// TIA Portal V17 export
// export: Created 2025-03-07T09:16:39.4097333Z, ExportSetting WithDefaults, DisplayName Totally Integrated Automation Portal, DisplayVersion V17 Update 8, DisplayName TIA Portal Openness, DisplayVersion V17 Update 8, DisplayName TIA Portal Version Control Interface, DisplayVersion V17, DisplayName SINAMICS Startdrive Advanced, DisplayVersion V17 SP2, DisplayName SINAMICS Startdrive G110M, G120, G120C, G120D, G120P, G115D, DisplayVersion V17 SP2, DisplayName SINAMICS Startdrive G130, G150, S120, S150, SINAMICS MV, S210, DisplayVersion V17 SP2, DisplayName STEP 7 Professional, DisplayVersion V17 Update 8, DisplayName SINUMERIK ONE STEP 7 Toolbox, DisplayVersion V17 Update 12, DisplayName SINUMERIK 840D sl STEP 7 Toolbox, DisplayVersion V17 Update 12, DisplayName STEP 7 Safety, DisplayVersion V17 Update 6, DisplayName WinCC Advanced, DisplayVersion V17 Update 8
FUNCTION "FC2420_CNC_PLC_SIGNALS" : Void   // FC2420, LAD
TITLE = NCK Inputs
{ S7_Optimized_Access := 'FALSE' }
AUTHOR : ETXETAR
VERSION : 1.0
// stored: AutoNumber false, IsIECCheckEnabled false, SetENOAutomatically false, UDAEnableTagReadback false
   VAR_TEMP
      ERROR : Bool;   // ERROR
      RESET_SIGNALS : Bool;   // RESET NC TO PLC SIGNALS
      ERROR_CODE : Int;   // ERROR CODE
      ZERO : Int;   // ZERO
   END_VAR
   VAR CONSTANT
      READ : Byte := 16#3;   // READ
      WRITE : Byte := 16#4;   // WRITE
   END_VAR
   VAR_TEMP   // added for the SCL form of the ladder/FBD networks
      _w1 : Bool;
   END_VAR
BEGIN

REGION Network 1: ZERO
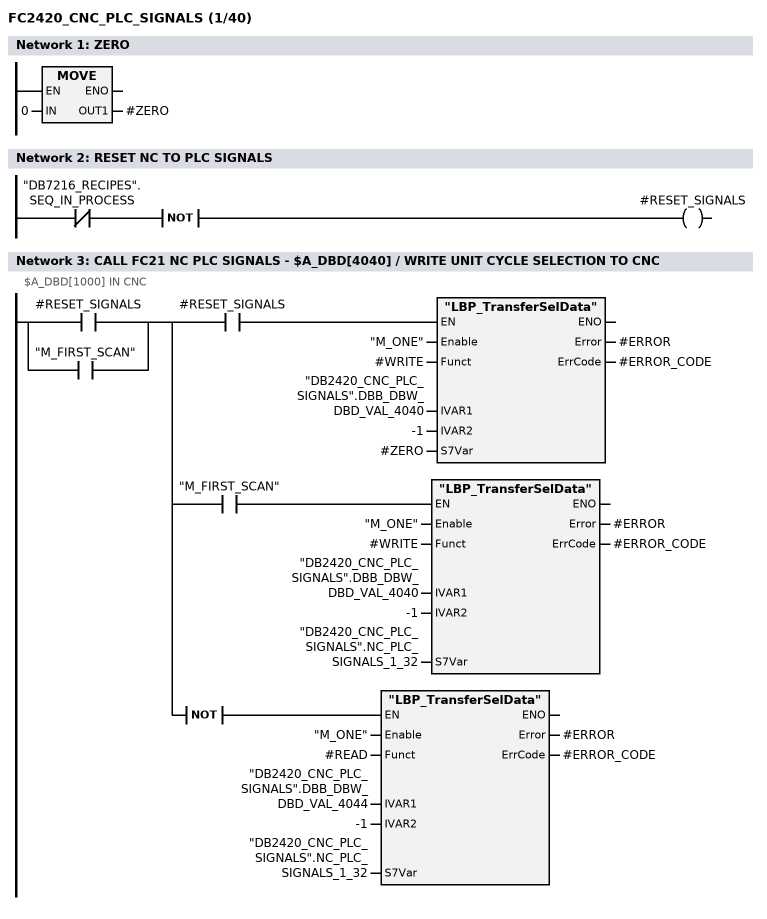
   RUNG wire#powerrail
      Move(in := 0, out1 => #ZERO)
   END_RUNG
   // the same network as SCL:
   #ZERO := 0;
END_REGION

REGION Network 2: RESET NC TO PLC SIGNALS
   RUNG wire#powerrail
      I_Contact( "DB7216_RECIPES".SEQ_IN_PROCESS )
      Not()
      Coil( #RESET_SIGNALS )
   END_RUNG
   // the same network as SCL:
   #RESET_SIGNALS := NOT (NOT "DB7216_RECIPES".SEQ_IN_PROCESS);
END_REGION

REGION Network 3: CALL FC21 NC PLC SIGNALS - $A_DBD[4040] / WRITE UNIT CYCLE SELECTION TO CNC
   // $A_DBD[1000] IN CNC
   RUNG wire#powerrail
      Contact( #RESET_SIGNALS )
      wire#w1
      Contact( #RESET_SIGNALS )
      "LBP_TransferSelData"(Enable := "M_ONE", Funct := #WRITE, IVAR1 := "DB2420_CNC_PLC_SIGNALS".DBB_DBW_DBD_VAL_4040, IVAR2 := -1, S7Var := #ZERO, Error => #ERROR, ErrCode => #ERROR_CODE)
   END_RUNG
   RUNG wire#powerrail
      Contact( "M_FIRST_SCAN" )
   END_RUNG wire#w1
   RUNG wire#w1
      Contact( "M_FIRST_SCAN" )
      "LBP_TransferSelData"(Enable := "M_ONE", Funct := #WRITE, IVAR1 := "DB2420_CNC_PLC_SIGNALS".DBB_DBW_DBD_VAL_4040, IVAR2 := -1, S7Var := "DB2420_CNC_PLC_SIGNALS".NC_PLC_SIGNALS_1_32, Error => #ERROR, ErrCode => #ERROR_CODE)
   END_RUNG
   RUNG wire#w1
      Not()
      "LBP_TransferSelData"(Enable := "M_ONE", Funct := #READ, IVAR1 := "DB2420_CNC_PLC_SIGNALS".DBB_DBW_DBD_VAL_4044, IVAR2 := -1, S7Var := "DB2420_CNC_PLC_SIGNALS".NC_PLC_SIGNALS_1_32, Error => #ERROR, ErrCode => #ERROR_CODE)
   END_RUNG
   // the same network as SCL:
   #_w1 := #RESET_SIGNALS OR "M_FIRST_SCAN";
   IF #_w1 AND #RESET_SIGNALS THEN
       "LBP_TransferSelData"(Enable := "M_ONE",
                             Funct := #WRITE,
                             IVAR1 := "DB2420_CNC_PLC_SIGNALS".DBB_DBW_DBD_VAL_4040,
                             IVAR2 := -1,
                             S7Var := #ZERO,
                             Error => #ERROR,
                             ErrCode => #ERROR_CODE);
   END_IF;
   IF #_w1 AND "M_FIRST_SCAN" THEN
       "LBP_TransferSelData"(Enable := "M_ONE",
                             Funct := #WRITE,
                             IVAR1 := "DB2420_CNC_PLC_SIGNALS".DBB_DBW_DBD_VAL_4040,
                             IVAR2 := -1,
                             S7Var := "DB2420_CNC_PLC_SIGNALS".NC_PLC_SIGNALS_1_32,
                             Error => #ERROR,
                             ErrCode => #ERROR_CODE);
   END_IF;
   IF NOT #_w1 THEN
       "LBP_TransferSelData"(Enable := "M_ONE",
                             Funct := #READ,
                             IVAR1 := "DB2420_CNC_PLC_SIGNALS".DBB_DBW_DBD_VAL_4044,
                             IVAR2 := -1,
                             S7Var := "DB2420_CNC_PLC_SIGNALS".NC_PLC_SIGNALS_1_32,
                             Error => #ERROR,
                             ErrCode => #ERROR_CODE);
   END_IF;
END_REGION

REGION Network 4: NC PLC SIGNALS 1-8
   // SIGNAL 1 -->  FIXTURE 1 CYLINDER 1 CLAMPED
   // SIGNAL 2 -->  FIXTURE 1 CYLINDER 2 CLAMPED
   // SIGNAL 3 -->  FIXTURE 1 CYLINDER 3 CLAMPED
   // SIGNAL 4 -->  FIXTURE 1 CYLINDER 4 CLAMPED
   // SIGNAL 5 -->  FIXTURE 1 CYLINDER 5 CLAMPED
   // SIGNAL 6 -->  FIXTURE 1 CYLINDER 6 CLAMPED
   // SIGNAL 7 -->  FIXTURE 1 CYLINDER 7 CLAMPED
   // SIGNAL 8 -->  FIXTURE 1 CYLINDER 8 CLAMPED
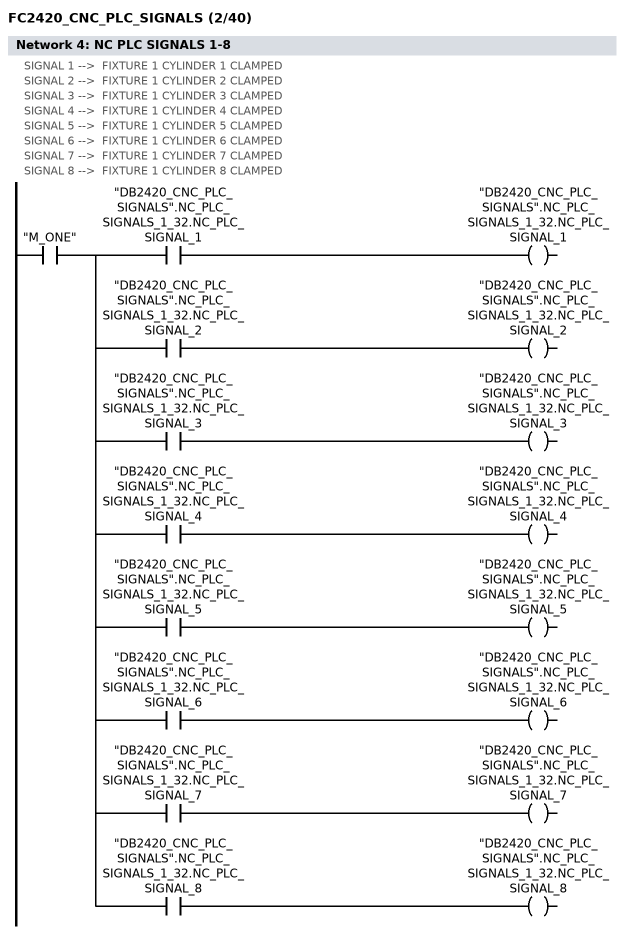
   RUNG wire#powerrail
      Contact( "M_ONE" )
      wire#w1
      Contact( "DB2420_CNC_PLC_SIGNALS".NC_PLC_SIGNALS_1_32.NC_PLC_SIGNAL_1 )
      Coil( "DB2420_CNC_PLC_SIGNALS".NC_PLC_SIGNALS_1_32.NC_PLC_SIGNAL_1 )
   END_RUNG
   RUNG wire#w1
      Contact( "DB2420_CNC_PLC_SIGNALS".NC_PLC_SIGNALS_1_32.NC_PLC_SIGNAL_2 )
      Coil( "DB2420_CNC_PLC_SIGNALS".NC_PLC_SIGNALS_1_32.NC_PLC_SIGNAL_2 )
   END_RUNG
   RUNG wire#w1
      Contact( "DB2420_CNC_PLC_SIGNALS".NC_PLC_SIGNALS_1_32.NC_PLC_SIGNAL_3 )
      Coil( "DB2420_CNC_PLC_SIGNALS".NC_PLC_SIGNALS_1_32.NC_PLC_SIGNAL_3 )
   END_RUNG
   RUNG wire#w1
      Contact( "DB2420_CNC_PLC_SIGNALS".NC_PLC_SIGNALS_1_32.NC_PLC_SIGNAL_4 )
      Coil( "DB2420_CNC_PLC_SIGNALS".NC_PLC_SIGNALS_1_32.NC_PLC_SIGNAL_4 )
   END_RUNG
   RUNG wire#w1
      Contact( "DB2420_CNC_PLC_SIGNALS".NC_PLC_SIGNALS_1_32.NC_PLC_SIGNAL_5 )
      Coil( "DB2420_CNC_PLC_SIGNALS".NC_PLC_SIGNALS_1_32.NC_PLC_SIGNAL_5 )
   END_RUNG
   RUNG wire#w1
      Contact( "DB2420_CNC_PLC_SIGNALS".NC_PLC_SIGNALS_1_32.NC_PLC_SIGNAL_6 )
      Coil( "DB2420_CNC_PLC_SIGNALS".NC_PLC_SIGNALS_1_32.NC_PLC_SIGNAL_6 )
   END_RUNG
   RUNG wire#w1
      Contact( "DB2420_CNC_PLC_SIGNALS".NC_PLC_SIGNALS_1_32.NC_PLC_SIGNAL_7 )
      Coil( "DB2420_CNC_PLC_SIGNALS".NC_PLC_SIGNALS_1_32.NC_PLC_SIGNAL_7 )
   END_RUNG
   RUNG wire#w1
      Contact( "DB2420_CNC_PLC_SIGNALS".NC_PLC_SIGNALS_1_32.NC_PLC_SIGNAL_8 )
      Coil( "DB2420_CNC_PLC_SIGNALS".NC_PLC_SIGNALS_1_32.NC_PLC_SIGNAL_8 )
   END_RUNG
   // the same network as SCL:
   "DB2420_CNC_PLC_SIGNALS".NC_PLC_SIGNALS_1_32.NC_PLC_SIGNAL_1 := "M_ONE" AND "DB2420_CNC_PLC_SIGNALS".NC_PLC_SIGNALS_1_32.NC_PLC_SIGNAL_1;
   "DB2420_CNC_PLC_SIGNALS".NC_PLC_SIGNALS_1_32.NC_PLC_SIGNAL_2 := "M_ONE" AND "DB2420_CNC_PLC_SIGNALS".NC_PLC_SIGNALS_1_32.NC_PLC_SIGNAL_2;
   "DB2420_CNC_PLC_SIGNALS".NC_PLC_SIGNALS_1_32.NC_PLC_SIGNAL_3 := "M_ONE" AND "DB2420_CNC_PLC_SIGNALS".NC_PLC_SIGNALS_1_32.NC_PLC_SIGNAL_3;
   "DB2420_CNC_PLC_SIGNALS".NC_PLC_SIGNALS_1_32.NC_PLC_SIGNAL_4 := "M_ONE" AND "DB2420_CNC_PLC_SIGNALS".NC_PLC_SIGNALS_1_32.NC_PLC_SIGNAL_4;
   "DB2420_CNC_PLC_SIGNALS".NC_PLC_SIGNALS_1_32.NC_PLC_SIGNAL_5 := "M_ONE" AND "DB2420_CNC_PLC_SIGNALS".NC_PLC_SIGNALS_1_32.NC_PLC_SIGNAL_5;
   "DB2420_CNC_PLC_SIGNALS".NC_PLC_SIGNALS_1_32.NC_PLC_SIGNAL_6 := "M_ONE" AND "DB2420_CNC_PLC_SIGNALS".NC_PLC_SIGNALS_1_32.NC_PLC_SIGNAL_6;
   "DB2420_CNC_PLC_SIGNALS".NC_PLC_SIGNALS_1_32.NC_PLC_SIGNAL_7 := "M_ONE" AND "DB2420_CNC_PLC_SIGNALS".NC_PLC_SIGNALS_1_32.NC_PLC_SIGNAL_7;
   "DB2420_CNC_PLC_SIGNALS".NC_PLC_SIGNALS_1_32.NC_PLC_SIGNAL_8 := "M_ONE" AND "DB2420_CNC_PLC_SIGNALS".NC_PLC_SIGNALS_1_32.NC_PLC_SIGNAL_8;
END_REGION

REGION Network 5: NC PLC SIGNALS 9-16
   // SIGNAL 9 -->  FIXTURE 1 CYLINDER 9 CLAMPED
   // SIGNAL 10 -->  FIXTURE 1 CYLINDER 10 CLAMPED
   // SIGNAL 11 -->  FIXTURE 1 CYLINDER 11 CLAMPED
   // SIGNAL 12 -->  FIXTURE 1 CYLINDER 12 CLAMPED
   // SIGNAL 13 -->  FIXTURE 1 CYLINDER 13 CLAMPED
   // SIGNAL 14 -->  FIXTURE 1 CYLINDER 14 CLAMPED
   // SIGNAL 15 -->  FIXTURE 1 CYLINDER 15 CLAMPED
   // SIGNAL 16 -->  FIXTURE 1 CYLINDER 16 CLAMPED
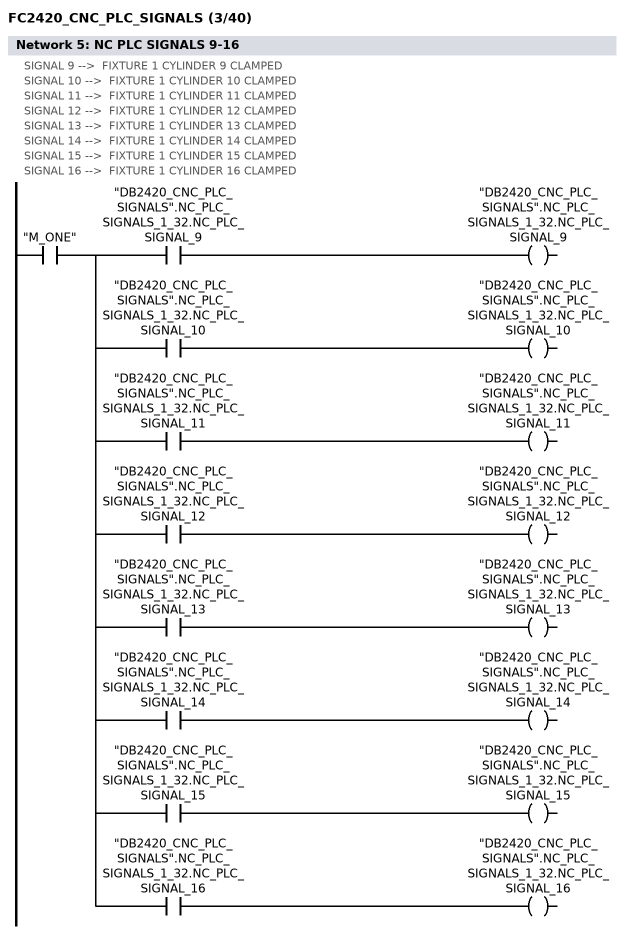
   RUNG wire#powerrail
      Contact( "M_ONE" )
      wire#w1
      Contact( "DB2420_CNC_PLC_SIGNALS".NC_PLC_SIGNALS_1_32.NC_PLC_SIGNAL_9 )
      Coil( "DB2420_CNC_PLC_SIGNALS".NC_PLC_SIGNALS_1_32.NC_PLC_SIGNAL_9 )
   END_RUNG
   RUNG wire#w1
      Contact( "DB2420_CNC_PLC_SIGNALS".NC_PLC_SIGNALS_1_32.NC_PLC_SIGNAL_10 )
      Coil( "DB2420_CNC_PLC_SIGNALS".NC_PLC_SIGNALS_1_32.NC_PLC_SIGNAL_10 )
   END_RUNG
   RUNG wire#w1
      Contact( "DB2420_CNC_PLC_SIGNALS".NC_PLC_SIGNALS_1_32.NC_PLC_SIGNAL_11 )
      Coil( "DB2420_CNC_PLC_SIGNALS".NC_PLC_SIGNALS_1_32.NC_PLC_SIGNAL_11 )
   END_RUNG
   RUNG wire#w1
      Contact( "DB2420_CNC_PLC_SIGNALS".NC_PLC_SIGNALS_1_32.NC_PLC_SIGNAL_12 )
      Coil( "DB2420_CNC_PLC_SIGNALS".NC_PLC_SIGNALS_1_32.NC_PLC_SIGNAL_12 )
   END_RUNG
   RUNG wire#w1
      Contact( "DB2420_CNC_PLC_SIGNALS".NC_PLC_SIGNALS_1_32.NC_PLC_SIGNAL_13 )
      Coil( "DB2420_CNC_PLC_SIGNALS".NC_PLC_SIGNALS_1_32.NC_PLC_SIGNAL_13 )
   END_RUNG
   RUNG wire#w1
      Contact( "DB2420_CNC_PLC_SIGNALS".NC_PLC_SIGNALS_1_32.NC_PLC_SIGNAL_14 )
      Coil( "DB2420_CNC_PLC_SIGNALS".NC_PLC_SIGNALS_1_32.NC_PLC_SIGNAL_14 )
   END_RUNG
   RUNG wire#w1
      Contact( "DB2420_CNC_PLC_SIGNALS".NC_PLC_SIGNALS_1_32.NC_PLC_SIGNAL_15 )
      Coil( "DB2420_CNC_PLC_SIGNALS".NC_PLC_SIGNALS_1_32.NC_PLC_SIGNAL_15 )
   END_RUNG
   RUNG wire#w1
      Contact( "DB2420_CNC_PLC_SIGNALS".NC_PLC_SIGNALS_1_32.NC_PLC_SIGNAL_16 )
      Coil( "DB2420_CNC_PLC_SIGNALS".NC_PLC_SIGNALS_1_32.NC_PLC_SIGNAL_16 )
   END_RUNG
   // the same network as SCL:
   "DB2420_CNC_PLC_SIGNALS".NC_PLC_SIGNALS_1_32.NC_PLC_SIGNAL_9 := "M_ONE" AND "DB2420_CNC_PLC_SIGNALS".NC_PLC_SIGNALS_1_32.NC_PLC_SIGNAL_9;
   "DB2420_CNC_PLC_SIGNALS".NC_PLC_SIGNALS_1_32.NC_PLC_SIGNAL_10 := "M_ONE" AND "DB2420_CNC_PLC_SIGNALS".NC_PLC_SIGNALS_1_32.NC_PLC_SIGNAL_10;
   "DB2420_CNC_PLC_SIGNALS".NC_PLC_SIGNALS_1_32.NC_PLC_SIGNAL_11 := "M_ONE" AND "DB2420_CNC_PLC_SIGNALS".NC_PLC_SIGNALS_1_32.NC_PLC_SIGNAL_11;
   "DB2420_CNC_PLC_SIGNALS".NC_PLC_SIGNALS_1_32.NC_PLC_SIGNAL_12 := "M_ONE" AND "DB2420_CNC_PLC_SIGNALS".NC_PLC_SIGNALS_1_32.NC_PLC_SIGNAL_12;
   "DB2420_CNC_PLC_SIGNALS".NC_PLC_SIGNALS_1_32.NC_PLC_SIGNAL_13 := "M_ONE" AND "DB2420_CNC_PLC_SIGNALS".NC_PLC_SIGNALS_1_32.NC_PLC_SIGNAL_13;
   "DB2420_CNC_PLC_SIGNALS".NC_PLC_SIGNALS_1_32.NC_PLC_SIGNAL_14 := "M_ONE" AND "DB2420_CNC_PLC_SIGNALS".NC_PLC_SIGNALS_1_32.NC_PLC_SIGNAL_14;
   "DB2420_CNC_PLC_SIGNALS".NC_PLC_SIGNALS_1_32.NC_PLC_SIGNAL_15 := "M_ONE" AND "DB2420_CNC_PLC_SIGNALS".NC_PLC_SIGNALS_1_32.NC_PLC_SIGNAL_15;
   "DB2420_CNC_PLC_SIGNALS".NC_PLC_SIGNALS_1_32.NC_PLC_SIGNAL_16 := "M_ONE" AND "DB2420_CNC_PLC_SIGNALS".NC_PLC_SIGNALS_1_32.NC_PLC_SIGNAL_16;
END_REGION

REGION Network 6: NC PLC SIGNALS 17-24
   // SIGNAL 17 -->  FIXTURE 1 CYLINDER 17 CLAMPED
   // SIGNAL 18 -->  FIXTURE 1 CYLINDER 18 CLAMPED
   // SIGNAL 19 -->  FIXTURE 1 CYLINDER 19 CLAMPED
   // SIGNAL 20 -->  FIXTURE 1 CYLINDER 20 CLAMPED
   // SIGNAL 21 -->  FIXTURE 1 CYLINDER 21 CLAMPED
   // SIGNAL 22 -->  FIXTURE 1 CYLINDER 22 CLAMPED
   // SIGNAL 23 -->  FIXTURE 1 CYLINDER 23 CLAMPED
   // SIGNAL 24 -->  FIXTURE 1 CYLINDER 24 CLAMPED
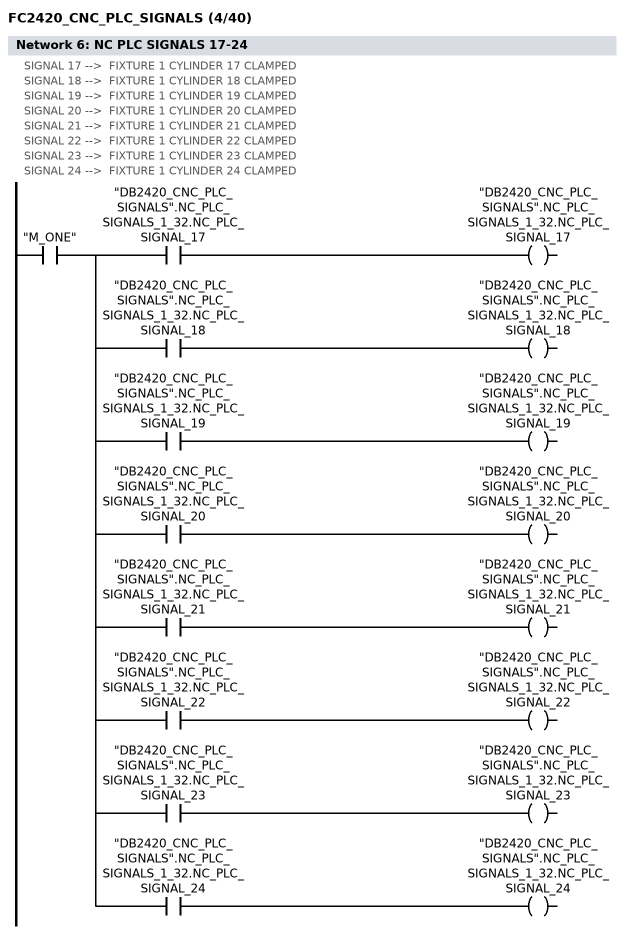
   RUNG wire#powerrail
      Contact( "M_ONE" )
      wire#w1
      Contact( "DB2420_CNC_PLC_SIGNALS".NC_PLC_SIGNALS_1_32.NC_PLC_SIGNAL_17 )
      Coil( "DB2420_CNC_PLC_SIGNALS".NC_PLC_SIGNALS_1_32.NC_PLC_SIGNAL_17 )
   END_RUNG
   RUNG wire#w1
      Contact( "DB2420_CNC_PLC_SIGNALS".NC_PLC_SIGNALS_1_32.NC_PLC_SIGNAL_18 )
      Coil( "DB2420_CNC_PLC_SIGNALS".NC_PLC_SIGNALS_1_32.NC_PLC_SIGNAL_18 )
   END_RUNG
   RUNG wire#w1
      Contact( "DB2420_CNC_PLC_SIGNALS".NC_PLC_SIGNALS_1_32.NC_PLC_SIGNAL_19 )
      Coil( "DB2420_CNC_PLC_SIGNALS".NC_PLC_SIGNALS_1_32.NC_PLC_SIGNAL_19 )
   END_RUNG
   RUNG wire#w1
      Contact( "DB2420_CNC_PLC_SIGNALS".NC_PLC_SIGNALS_1_32.NC_PLC_SIGNAL_20 )
      Coil( "DB2420_CNC_PLC_SIGNALS".NC_PLC_SIGNALS_1_32.NC_PLC_SIGNAL_20 )
   END_RUNG
   RUNG wire#w1
      Contact( "DB2420_CNC_PLC_SIGNALS".NC_PLC_SIGNALS_1_32.NC_PLC_SIGNAL_21 )
      Coil( "DB2420_CNC_PLC_SIGNALS".NC_PLC_SIGNALS_1_32.NC_PLC_SIGNAL_21 )
   END_RUNG
   RUNG wire#w1
      Contact( "DB2420_CNC_PLC_SIGNALS".NC_PLC_SIGNALS_1_32.NC_PLC_SIGNAL_22 )
      Coil( "DB2420_CNC_PLC_SIGNALS".NC_PLC_SIGNALS_1_32.NC_PLC_SIGNAL_22 )
   END_RUNG
   RUNG wire#w1
      Contact( "DB2420_CNC_PLC_SIGNALS".NC_PLC_SIGNALS_1_32.NC_PLC_SIGNAL_23 )
      Coil( "DB2420_CNC_PLC_SIGNALS".NC_PLC_SIGNALS_1_32.NC_PLC_SIGNAL_23 )
   END_RUNG
   RUNG wire#w1
      Contact( "DB2420_CNC_PLC_SIGNALS".NC_PLC_SIGNALS_1_32.NC_PLC_SIGNAL_24 )
      Coil( "DB2420_CNC_PLC_SIGNALS".NC_PLC_SIGNALS_1_32.NC_PLC_SIGNAL_24 )
   END_RUNG
   // the same network as SCL:
   "DB2420_CNC_PLC_SIGNALS".NC_PLC_SIGNALS_1_32.NC_PLC_SIGNAL_17 := "M_ONE" AND "DB2420_CNC_PLC_SIGNALS".NC_PLC_SIGNALS_1_32.NC_PLC_SIGNAL_17;
   "DB2420_CNC_PLC_SIGNALS".NC_PLC_SIGNALS_1_32.NC_PLC_SIGNAL_18 := "M_ONE" AND "DB2420_CNC_PLC_SIGNALS".NC_PLC_SIGNALS_1_32.NC_PLC_SIGNAL_18;
   "DB2420_CNC_PLC_SIGNALS".NC_PLC_SIGNALS_1_32.NC_PLC_SIGNAL_19 := "M_ONE" AND "DB2420_CNC_PLC_SIGNALS".NC_PLC_SIGNALS_1_32.NC_PLC_SIGNAL_19;
   "DB2420_CNC_PLC_SIGNALS".NC_PLC_SIGNALS_1_32.NC_PLC_SIGNAL_20 := "M_ONE" AND "DB2420_CNC_PLC_SIGNALS".NC_PLC_SIGNALS_1_32.NC_PLC_SIGNAL_20;
   "DB2420_CNC_PLC_SIGNALS".NC_PLC_SIGNALS_1_32.NC_PLC_SIGNAL_21 := "M_ONE" AND "DB2420_CNC_PLC_SIGNALS".NC_PLC_SIGNALS_1_32.NC_PLC_SIGNAL_21;
   "DB2420_CNC_PLC_SIGNALS".NC_PLC_SIGNALS_1_32.NC_PLC_SIGNAL_22 := "M_ONE" AND "DB2420_CNC_PLC_SIGNALS".NC_PLC_SIGNALS_1_32.NC_PLC_SIGNAL_22;
   "DB2420_CNC_PLC_SIGNALS".NC_PLC_SIGNALS_1_32.NC_PLC_SIGNAL_23 := "M_ONE" AND "DB2420_CNC_PLC_SIGNALS".NC_PLC_SIGNALS_1_32.NC_PLC_SIGNAL_23;
   "DB2420_CNC_PLC_SIGNALS".NC_PLC_SIGNALS_1_32.NC_PLC_SIGNAL_24 := "M_ONE" AND "DB2420_CNC_PLC_SIGNALS".NC_PLC_SIGNALS_1_32.NC_PLC_SIGNAL_24;
END_REGION

REGION Network 7: NC PLC SIGNALS 25-32
   // SIGNAL 25 -->  FIXTURE 1 CYLINDER 1 UNCLAMPED
   // SIGNAL 26 -->  FIXTURE 1 CYLINDER 2 UNCLAMPED
   // SIGNAL 27 -->  FIXTURE 1 CYLINDER 3 UNCLAMPED
   // SIGNAL 28 -->  FIXTURE 1 CYLINDER 4 UNCLAMPED
   // SIGNAL 29 -->  FIXTURE 1 CYLINDER 5 UNCLAMPED
   // SIGNAL 30 -->  FIXTURE 1 CYLINDER 6 UNCLAMPED
   // SIGNAL 31 -->  FIXTURE 1 CYLINDER 7 UNCLAMPED
   // SIGNAL 32 -->  FIXTURE 1 CYLINDER 8 UNCLAMPED
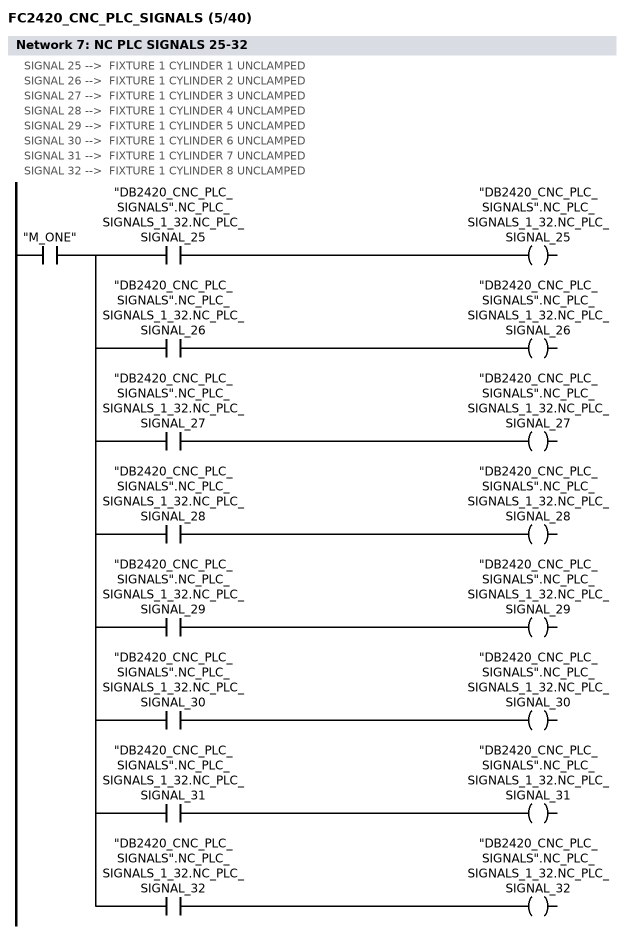
   RUNG wire#powerrail
      Contact( "M_ONE" )
      wire#w1
      Contact( "DB2420_CNC_PLC_SIGNALS".NC_PLC_SIGNALS_1_32.NC_PLC_SIGNAL_25 )
      Coil( "DB2420_CNC_PLC_SIGNALS".NC_PLC_SIGNALS_1_32.NC_PLC_SIGNAL_25 )
   END_RUNG
   RUNG wire#w1
      Contact( "DB2420_CNC_PLC_SIGNALS".NC_PLC_SIGNALS_1_32.NC_PLC_SIGNAL_26 )
      Coil( "DB2420_CNC_PLC_SIGNALS".NC_PLC_SIGNALS_1_32.NC_PLC_SIGNAL_26 )
   END_RUNG
   RUNG wire#w1
      Contact( "DB2420_CNC_PLC_SIGNALS".NC_PLC_SIGNALS_1_32.NC_PLC_SIGNAL_27 )
      Coil( "DB2420_CNC_PLC_SIGNALS".NC_PLC_SIGNALS_1_32.NC_PLC_SIGNAL_27 )
   END_RUNG
   RUNG wire#w1
      Contact( "DB2420_CNC_PLC_SIGNALS".NC_PLC_SIGNALS_1_32.NC_PLC_SIGNAL_28 )
      Coil( "DB2420_CNC_PLC_SIGNALS".NC_PLC_SIGNALS_1_32.NC_PLC_SIGNAL_28 )
   END_RUNG
   RUNG wire#w1
      Contact( "DB2420_CNC_PLC_SIGNALS".NC_PLC_SIGNALS_1_32.NC_PLC_SIGNAL_29 )
      Coil( "DB2420_CNC_PLC_SIGNALS".NC_PLC_SIGNALS_1_32.NC_PLC_SIGNAL_29 )
   END_RUNG
   RUNG wire#w1
      Contact( "DB2420_CNC_PLC_SIGNALS".NC_PLC_SIGNALS_1_32.NC_PLC_SIGNAL_30 )
      Coil( "DB2420_CNC_PLC_SIGNALS".NC_PLC_SIGNALS_1_32.NC_PLC_SIGNAL_30 )
   END_RUNG
   RUNG wire#w1
      Contact( "DB2420_CNC_PLC_SIGNALS".NC_PLC_SIGNALS_1_32.NC_PLC_SIGNAL_31 )
      Coil( "DB2420_CNC_PLC_SIGNALS".NC_PLC_SIGNALS_1_32.NC_PLC_SIGNAL_31 )
   END_RUNG
   RUNG wire#w1
      Contact( "DB2420_CNC_PLC_SIGNALS".NC_PLC_SIGNALS_1_32.NC_PLC_SIGNAL_32 )
      Coil( "DB2420_CNC_PLC_SIGNALS".NC_PLC_SIGNALS_1_32.NC_PLC_SIGNAL_32 )
   END_RUNG
   // the same network as SCL:
   "DB2420_CNC_PLC_SIGNALS".NC_PLC_SIGNALS_1_32.NC_PLC_SIGNAL_25 := "M_ONE" AND "DB2420_CNC_PLC_SIGNALS".NC_PLC_SIGNALS_1_32.NC_PLC_SIGNAL_25;
   "DB2420_CNC_PLC_SIGNALS".NC_PLC_SIGNALS_1_32.NC_PLC_SIGNAL_26 := "M_ONE" AND "DB2420_CNC_PLC_SIGNALS".NC_PLC_SIGNALS_1_32.NC_PLC_SIGNAL_26;
   "DB2420_CNC_PLC_SIGNALS".NC_PLC_SIGNALS_1_32.NC_PLC_SIGNAL_27 := "M_ONE" AND "DB2420_CNC_PLC_SIGNALS".NC_PLC_SIGNALS_1_32.NC_PLC_SIGNAL_27;
   "DB2420_CNC_PLC_SIGNALS".NC_PLC_SIGNALS_1_32.NC_PLC_SIGNAL_28 := "M_ONE" AND "DB2420_CNC_PLC_SIGNALS".NC_PLC_SIGNALS_1_32.NC_PLC_SIGNAL_28;
   "DB2420_CNC_PLC_SIGNALS".NC_PLC_SIGNALS_1_32.NC_PLC_SIGNAL_29 := "M_ONE" AND "DB2420_CNC_PLC_SIGNALS".NC_PLC_SIGNALS_1_32.NC_PLC_SIGNAL_29;
   "DB2420_CNC_PLC_SIGNALS".NC_PLC_SIGNALS_1_32.NC_PLC_SIGNAL_30 := "M_ONE" AND "DB2420_CNC_PLC_SIGNALS".NC_PLC_SIGNALS_1_32.NC_PLC_SIGNAL_30;
   "DB2420_CNC_PLC_SIGNALS".NC_PLC_SIGNALS_1_32.NC_PLC_SIGNAL_31 := "M_ONE" AND "DB2420_CNC_PLC_SIGNALS".NC_PLC_SIGNALS_1_32.NC_PLC_SIGNAL_31;
   "DB2420_CNC_PLC_SIGNALS".NC_PLC_SIGNALS_1_32.NC_PLC_SIGNAL_32 := "M_ONE" AND "DB2420_CNC_PLC_SIGNALS".NC_PLC_SIGNALS_1_32.NC_PLC_SIGNAL_32;
END_REGION

REGION Network 8: CALL FC21 NC PLC SIGNALS- $A_DBD[4044] / WRITE UNIT CYCLE SELECTION TO CNC
   // $A_DBD[1000] IN CNC
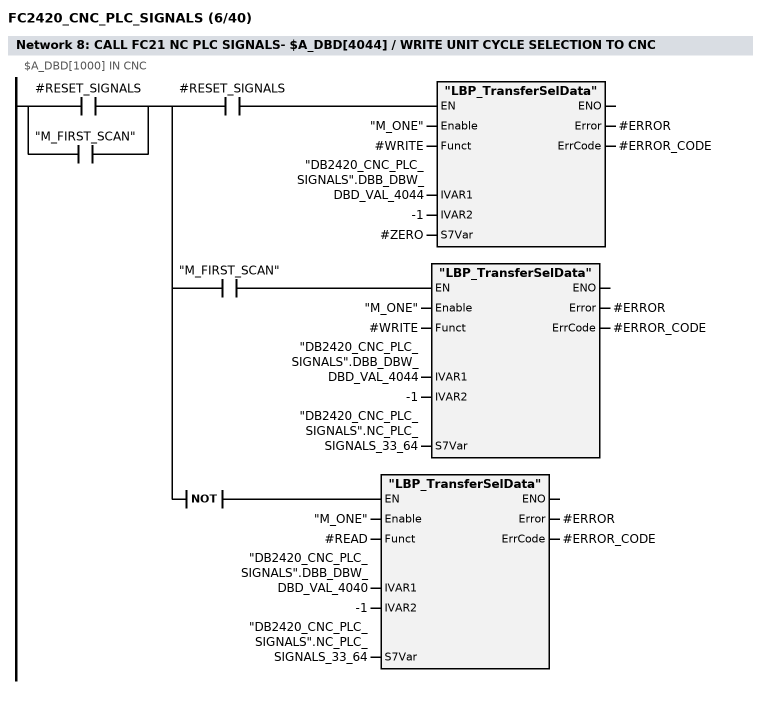
   RUNG wire#powerrail
      Contact( #RESET_SIGNALS )
      wire#w1
      Contact( #RESET_SIGNALS )
      "LBP_TransferSelData"(Enable := "M_ONE", Funct := #WRITE, IVAR1 := "DB2420_CNC_PLC_SIGNALS".DBB_DBW_DBD_VAL_4044, IVAR2 := -1, S7Var := #ZERO, Error => #ERROR, ErrCode => #ERROR_CODE)
   END_RUNG
   RUNG wire#powerrail
      Contact( "M_FIRST_SCAN" )
   END_RUNG wire#w1
   RUNG wire#w1
      Contact( "M_FIRST_SCAN" )
      "LBP_TransferSelData"(Enable := "M_ONE", Funct := #WRITE, IVAR1 := "DB2420_CNC_PLC_SIGNALS".DBB_DBW_DBD_VAL_4044, IVAR2 := -1, S7Var := "DB2420_CNC_PLC_SIGNALS".NC_PLC_SIGNALS_33_64, Error => #ERROR, ErrCode => #ERROR_CODE)
   END_RUNG
   RUNG wire#w1
      Not()
      "LBP_TransferSelData"(Enable := "M_ONE", Funct := #READ, IVAR1 := "DB2420_CNC_PLC_SIGNALS".DBB_DBW_DBD_VAL_4040, IVAR2 := -1, S7Var := "DB2420_CNC_PLC_SIGNALS".NC_PLC_SIGNALS_33_64, Error => #ERROR, ErrCode => #ERROR_CODE)
   END_RUNG
   // the same network as SCL:
   #_w1 := #RESET_SIGNALS OR "M_FIRST_SCAN";
   IF #_w1 AND #RESET_SIGNALS THEN
       "LBP_TransferSelData"(Enable := "M_ONE",
                             Funct := #WRITE,
                             IVAR1 := "DB2420_CNC_PLC_SIGNALS".DBB_DBW_DBD_VAL_4044,
                             IVAR2 := -1,
                             S7Var := #ZERO,
                             Error => #ERROR,
                             ErrCode => #ERROR_CODE);
   END_IF;
   IF #_w1 AND "M_FIRST_SCAN" THEN
       "LBP_TransferSelData"(Enable := "M_ONE",
                             Funct := #WRITE,
                             IVAR1 := "DB2420_CNC_PLC_SIGNALS".DBB_DBW_DBD_VAL_4044,
                             IVAR2 := -1,
                             S7Var := "DB2420_CNC_PLC_SIGNALS".NC_PLC_SIGNALS_33_64,
                             Error => #ERROR,
                             ErrCode => #ERROR_CODE);
   END_IF;
   IF NOT #_w1 THEN
       "LBP_TransferSelData"(Enable := "M_ONE",
                             Funct := #READ,
                             IVAR1 := "DB2420_CNC_PLC_SIGNALS".DBB_DBW_DBD_VAL_4040,
                             IVAR2 := -1,
                             S7Var := "DB2420_CNC_PLC_SIGNALS".NC_PLC_SIGNALS_33_64,
                             Error => #ERROR,
                             ErrCode => #ERROR_CODE);
   END_IF;
END_REGION

REGION Network 9: NC PLC SIGNALS 33-40
   // SIGNAL 33 -->  FIXTURE 1 CYLINDER 9 UNCLAMPED
   // SIGNAL 34 -->  FIXTURE 1 CYLINDER 10 UNCLAMPED
   // SIGNAL 35 -->  FIXTURE 1 CYLINDER 11 UNCLAMPED
   // SIGNAL 36 -->  FIXTURE 1 CYLINDER 12 UNCLAMPED
   // SIGNAL 37 -->  FIXTURE 1 CYLINDER 13 UNCLAMPED
   // SIGNAL 38 -->  FIXTURE 1 CYLINDER 14 UNCLAMPED
   // SIGNAL 39 -->  FIXTURE 1 CYLINDER 15 UNCLAMPED
   // SIGNAL 40 -->  FIXTURE 1 CYLINDER 16 UNCLAMPED
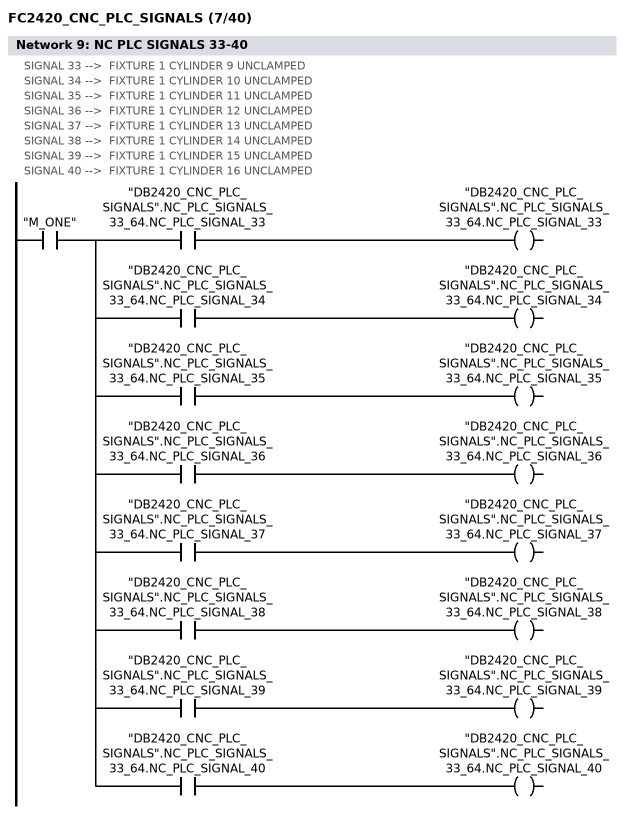
   RUNG wire#powerrail
      Contact( "M_ONE" )
      wire#w1
      Contact( "DB2420_CNC_PLC_SIGNALS".NC_PLC_SIGNALS_33_64.NC_PLC_SIGNAL_33 )
      Coil( "DB2420_CNC_PLC_SIGNALS".NC_PLC_SIGNALS_33_64.NC_PLC_SIGNAL_33 )
   END_RUNG
   RUNG wire#w1
      Contact( "DB2420_CNC_PLC_SIGNALS".NC_PLC_SIGNALS_33_64.NC_PLC_SIGNAL_34 )
      Coil( "DB2420_CNC_PLC_SIGNALS".NC_PLC_SIGNALS_33_64.NC_PLC_SIGNAL_34 )
   END_RUNG
   RUNG wire#w1
      Contact( "DB2420_CNC_PLC_SIGNALS".NC_PLC_SIGNALS_33_64.NC_PLC_SIGNAL_35 )
      Coil( "DB2420_CNC_PLC_SIGNALS".NC_PLC_SIGNALS_33_64.NC_PLC_SIGNAL_35 )
   END_RUNG
   RUNG wire#w1
      Contact( "DB2420_CNC_PLC_SIGNALS".NC_PLC_SIGNALS_33_64.NC_PLC_SIGNAL_36 )
      Coil( "DB2420_CNC_PLC_SIGNALS".NC_PLC_SIGNALS_33_64.NC_PLC_SIGNAL_36 )
   END_RUNG
   RUNG wire#w1
      Contact( "DB2420_CNC_PLC_SIGNALS".NC_PLC_SIGNALS_33_64.NC_PLC_SIGNAL_37 )
      Coil( "DB2420_CNC_PLC_SIGNALS".NC_PLC_SIGNALS_33_64.NC_PLC_SIGNAL_37 )
   END_RUNG
   RUNG wire#w1
      Contact( "DB2420_CNC_PLC_SIGNALS".NC_PLC_SIGNALS_33_64.NC_PLC_SIGNAL_38 )
      Coil( "DB2420_CNC_PLC_SIGNALS".NC_PLC_SIGNALS_33_64.NC_PLC_SIGNAL_38 )
   END_RUNG
   RUNG wire#w1
      Contact( "DB2420_CNC_PLC_SIGNALS".NC_PLC_SIGNALS_33_64.NC_PLC_SIGNAL_39 )
      Coil( "DB2420_CNC_PLC_SIGNALS".NC_PLC_SIGNALS_33_64.NC_PLC_SIGNAL_39 )
   END_RUNG
   RUNG wire#w1
      Contact( "DB2420_CNC_PLC_SIGNALS".NC_PLC_SIGNALS_33_64.NC_PLC_SIGNAL_40 )
      Coil( "DB2420_CNC_PLC_SIGNALS".NC_PLC_SIGNALS_33_64.NC_PLC_SIGNAL_40 )
   END_RUNG
   // the same network as SCL:
   "DB2420_CNC_PLC_SIGNALS".NC_PLC_SIGNALS_33_64.NC_PLC_SIGNAL_33 := "M_ONE" AND "DB2420_CNC_PLC_SIGNALS".NC_PLC_SIGNALS_33_64.NC_PLC_SIGNAL_33;
   "DB2420_CNC_PLC_SIGNALS".NC_PLC_SIGNALS_33_64.NC_PLC_SIGNAL_34 := "M_ONE" AND "DB2420_CNC_PLC_SIGNALS".NC_PLC_SIGNALS_33_64.NC_PLC_SIGNAL_34;
   "DB2420_CNC_PLC_SIGNALS".NC_PLC_SIGNALS_33_64.NC_PLC_SIGNAL_35 := "M_ONE" AND "DB2420_CNC_PLC_SIGNALS".NC_PLC_SIGNALS_33_64.NC_PLC_SIGNAL_35;
   "DB2420_CNC_PLC_SIGNALS".NC_PLC_SIGNALS_33_64.NC_PLC_SIGNAL_36 := "M_ONE" AND "DB2420_CNC_PLC_SIGNALS".NC_PLC_SIGNALS_33_64.NC_PLC_SIGNAL_36;
   "DB2420_CNC_PLC_SIGNALS".NC_PLC_SIGNALS_33_64.NC_PLC_SIGNAL_37 := "M_ONE" AND "DB2420_CNC_PLC_SIGNALS".NC_PLC_SIGNALS_33_64.NC_PLC_SIGNAL_37;
   "DB2420_CNC_PLC_SIGNALS".NC_PLC_SIGNALS_33_64.NC_PLC_SIGNAL_38 := "M_ONE" AND "DB2420_CNC_PLC_SIGNALS".NC_PLC_SIGNALS_33_64.NC_PLC_SIGNAL_38;
   "DB2420_CNC_PLC_SIGNALS".NC_PLC_SIGNALS_33_64.NC_PLC_SIGNAL_39 := "M_ONE" AND "DB2420_CNC_PLC_SIGNALS".NC_PLC_SIGNALS_33_64.NC_PLC_SIGNAL_39;
   "DB2420_CNC_PLC_SIGNALS".NC_PLC_SIGNALS_33_64.NC_PLC_SIGNAL_40 := "M_ONE" AND "DB2420_CNC_PLC_SIGNALS".NC_PLC_SIGNALS_33_64.NC_PLC_SIGNAL_40;
END_REGION

REGION Network 10: NC PLC SIGNALS 41-48
   // SIGNAL 41 -->  FIXTURE 1 CYLINDER 17 UNCLAMPED
   // SIGNAL 42 -->  FIXTURE 1 CYLINDER 18 UNCLAMPED
   // SIGNAL 43 -->  FIXTURE 1 CYLINDER 19 UNCLAMPED
   // SIGNAL 44 -->  FIXTURE 1 CYLINDER 20 UNCLAMPED
   // SIGNAL 45 -->  FIXTURE 1 CYLINDER 21 UNCLAMPED
   // SIGNAL 46 -->  FIXTURE 1 CYLINDER 22 UNCLAMPED
   // SIGNAL 47 -->  FIXTURE 1 CYLINDER 23 UNCLAMPED
   // SIGNAL 48 -->  FIXTURE 1 CYLINDER 24 UNCLAMPED
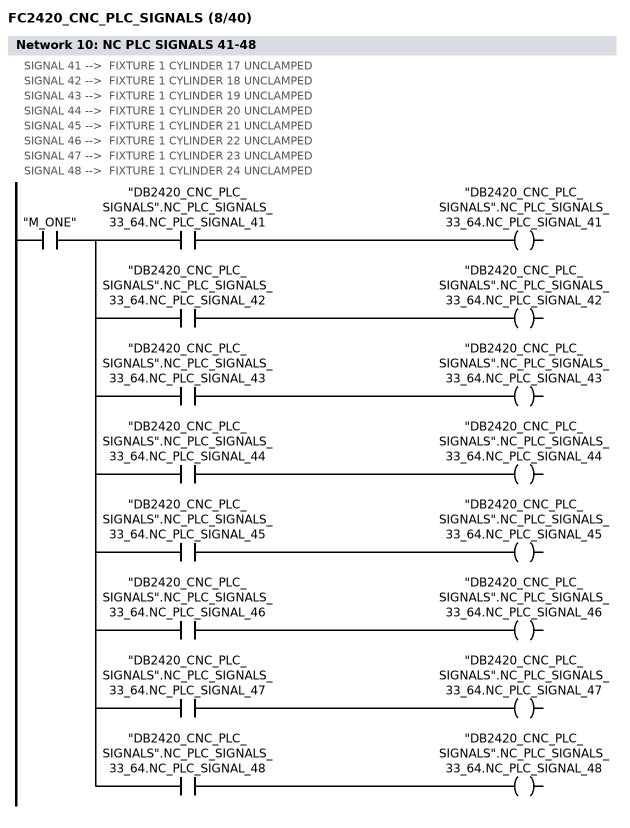
   RUNG wire#powerrail
      Contact( "M_ONE" )
      wire#w1
      Contact( "DB2420_CNC_PLC_SIGNALS".NC_PLC_SIGNALS_33_64.NC_PLC_SIGNAL_41 )
      Coil( "DB2420_CNC_PLC_SIGNALS".NC_PLC_SIGNALS_33_64.NC_PLC_SIGNAL_41 )
   END_RUNG
   RUNG wire#w1
      Contact( "DB2420_CNC_PLC_SIGNALS".NC_PLC_SIGNALS_33_64.NC_PLC_SIGNAL_42 )
      Coil( "DB2420_CNC_PLC_SIGNALS".NC_PLC_SIGNALS_33_64.NC_PLC_SIGNAL_42 )
   END_RUNG
   RUNG wire#w1
      Contact( "DB2420_CNC_PLC_SIGNALS".NC_PLC_SIGNALS_33_64.NC_PLC_SIGNAL_43 )
      Coil( "DB2420_CNC_PLC_SIGNALS".NC_PLC_SIGNALS_33_64.NC_PLC_SIGNAL_43 )
   END_RUNG
   RUNG wire#w1
      Contact( "DB2420_CNC_PLC_SIGNALS".NC_PLC_SIGNALS_33_64.NC_PLC_SIGNAL_44 )
      Coil( "DB2420_CNC_PLC_SIGNALS".NC_PLC_SIGNALS_33_64.NC_PLC_SIGNAL_44 )
   END_RUNG
   RUNG wire#w1
      Contact( "DB2420_CNC_PLC_SIGNALS".NC_PLC_SIGNALS_33_64.NC_PLC_SIGNAL_45 )
      Coil( "DB2420_CNC_PLC_SIGNALS".NC_PLC_SIGNALS_33_64.NC_PLC_SIGNAL_45 )
   END_RUNG
   RUNG wire#w1
      Contact( "DB2420_CNC_PLC_SIGNALS".NC_PLC_SIGNALS_33_64.NC_PLC_SIGNAL_46 )
      Coil( "DB2420_CNC_PLC_SIGNALS".NC_PLC_SIGNALS_33_64.NC_PLC_SIGNAL_46 )
   END_RUNG
   RUNG wire#w1
      Contact( "DB2420_CNC_PLC_SIGNALS".NC_PLC_SIGNALS_33_64.NC_PLC_SIGNAL_47 )
      Coil( "DB2420_CNC_PLC_SIGNALS".NC_PLC_SIGNALS_33_64.NC_PLC_SIGNAL_47 )
   END_RUNG
   RUNG wire#w1
      Contact( "DB2420_CNC_PLC_SIGNALS".NC_PLC_SIGNALS_33_64.NC_PLC_SIGNAL_48 )
      Coil( "DB2420_CNC_PLC_SIGNALS".NC_PLC_SIGNALS_33_64.NC_PLC_SIGNAL_48 )
   END_RUNG
   // the same network as SCL:
   "DB2420_CNC_PLC_SIGNALS".NC_PLC_SIGNALS_33_64.NC_PLC_SIGNAL_41 := "M_ONE" AND "DB2420_CNC_PLC_SIGNALS".NC_PLC_SIGNALS_33_64.NC_PLC_SIGNAL_41;
   "DB2420_CNC_PLC_SIGNALS".NC_PLC_SIGNALS_33_64.NC_PLC_SIGNAL_42 := "M_ONE" AND "DB2420_CNC_PLC_SIGNALS".NC_PLC_SIGNALS_33_64.NC_PLC_SIGNAL_42;
   "DB2420_CNC_PLC_SIGNALS".NC_PLC_SIGNALS_33_64.NC_PLC_SIGNAL_43 := "M_ONE" AND "DB2420_CNC_PLC_SIGNALS".NC_PLC_SIGNALS_33_64.NC_PLC_SIGNAL_43;
   "DB2420_CNC_PLC_SIGNALS".NC_PLC_SIGNALS_33_64.NC_PLC_SIGNAL_44 := "M_ONE" AND "DB2420_CNC_PLC_SIGNALS".NC_PLC_SIGNALS_33_64.NC_PLC_SIGNAL_44;
   "DB2420_CNC_PLC_SIGNALS".NC_PLC_SIGNALS_33_64.NC_PLC_SIGNAL_45 := "M_ONE" AND "DB2420_CNC_PLC_SIGNALS".NC_PLC_SIGNALS_33_64.NC_PLC_SIGNAL_45;
   "DB2420_CNC_PLC_SIGNALS".NC_PLC_SIGNALS_33_64.NC_PLC_SIGNAL_46 := "M_ONE" AND "DB2420_CNC_PLC_SIGNALS".NC_PLC_SIGNALS_33_64.NC_PLC_SIGNAL_46;
   "DB2420_CNC_PLC_SIGNALS".NC_PLC_SIGNALS_33_64.NC_PLC_SIGNAL_47 := "M_ONE" AND "DB2420_CNC_PLC_SIGNALS".NC_PLC_SIGNALS_33_64.NC_PLC_SIGNAL_47;
   "DB2420_CNC_PLC_SIGNALS".NC_PLC_SIGNALS_33_64.NC_PLC_SIGNAL_48 := "M_ONE" AND "DB2420_CNC_PLC_SIGNALS".NC_PLC_SIGNALS_33_64.NC_PLC_SIGNAL_48;
END_REGION

REGION Network 11: NC PLC SIGNALS 49-56
   // SIGNAL 49 -->  FIXTURE 2 CYLINDER 1 CLAMPED
   // SIGNAL 50 -->  FIXTURE 2 CYLINDER 2 CLAMPED
   // SIGNAL 51 -->   FIXTURE 2 CYLINDER 3 CLAMPED
   // SIGNAL 52 -->   FIXTURE 2 CYLINDER 4 CLAMPED
   // SIGNAL 53 -->   FIXTURE 2 CYLINDER 5 CLAMPED
   // SIGNAL 54 -->   FIXTURE 2 CYLINDER 6 CLAMPED
   // SIGNAL 55 -->   FIXTURE 2 CYLINDER 7 CLAMPED
   // SIGNAL 56 -->   FIXTURE 2 CYLINDER 8 CLAMPED
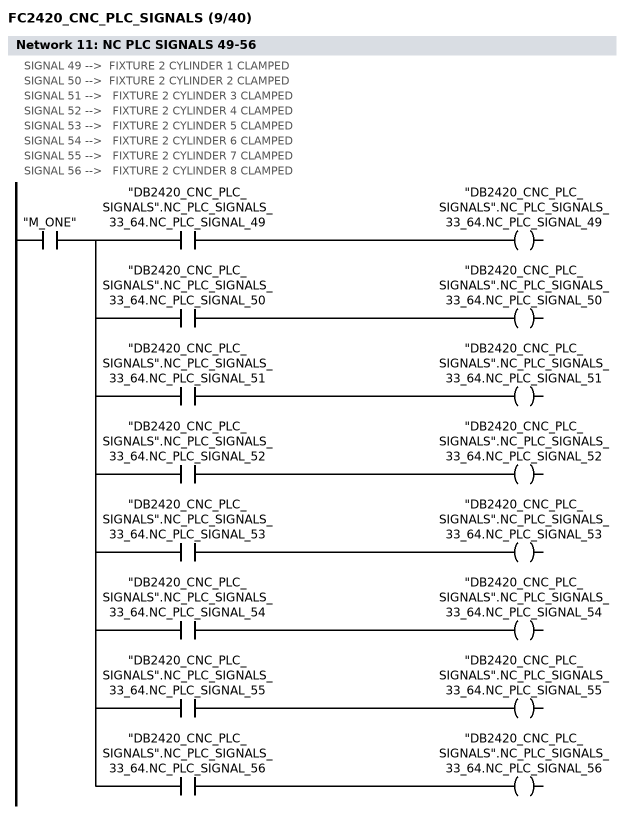
   RUNG wire#powerrail
      Contact( "M_ONE" )
      wire#w1
      Contact( "DB2420_CNC_PLC_SIGNALS".NC_PLC_SIGNALS_33_64.NC_PLC_SIGNAL_49 )
      Coil( "DB2420_CNC_PLC_SIGNALS".NC_PLC_SIGNALS_33_64.NC_PLC_SIGNAL_49 )
   END_RUNG
   RUNG wire#w1
      Contact( "DB2420_CNC_PLC_SIGNALS".NC_PLC_SIGNALS_33_64.NC_PLC_SIGNAL_50 )
      Coil( "DB2420_CNC_PLC_SIGNALS".NC_PLC_SIGNALS_33_64.NC_PLC_SIGNAL_50 )
   END_RUNG
   RUNG wire#w1
      Contact( "DB2420_CNC_PLC_SIGNALS".NC_PLC_SIGNALS_33_64.NC_PLC_SIGNAL_51 )
      Coil( "DB2420_CNC_PLC_SIGNALS".NC_PLC_SIGNALS_33_64.NC_PLC_SIGNAL_51 )
   END_RUNG
   RUNG wire#w1
      Contact( "DB2420_CNC_PLC_SIGNALS".NC_PLC_SIGNALS_33_64.NC_PLC_SIGNAL_52 )
      Coil( "DB2420_CNC_PLC_SIGNALS".NC_PLC_SIGNALS_33_64.NC_PLC_SIGNAL_52 )
   END_RUNG
   RUNG wire#w1
      Contact( "DB2420_CNC_PLC_SIGNALS".NC_PLC_SIGNALS_33_64.NC_PLC_SIGNAL_53 )
      Coil( "DB2420_CNC_PLC_SIGNALS".NC_PLC_SIGNALS_33_64.NC_PLC_SIGNAL_53 )
   END_RUNG
   RUNG wire#w1
      Contact( "DB2420_CNC_PLC_SIGNALS".NC_PLC_SIGNALS_33_64.NC_PLC_SIGNAL_54 )
      Coil( "DB2420_CNC_PLC_SIGNALS".NC_PLC_SIGNALS_33_64.NC_PLC_SIGNAL_54 )
   END_RUNG
   RUNG wire#w1
      Contact( "DB2420_CNC_PLC_SIGNALS".NC_PLC_SIGNALS_33_64.NC_PLC_SIGNAL_55 )
      Coil( "DB2420_CNC_PLC_SIGNALS".NC_PLC_SIGNALS_33_64.NC_PLC_SIGNAL_55 )
   END_RUNG
   RUNG wire#w1
      Contact( "DB2420_CNC_PLC_SIGNALS".NC_PLC_SIGNALS_33_64.NC_PLC_SIGNAL_56 )
      Coil( "DB2420_CNC_PLC_SIGNALS".NC_PLC_SIGNALS_33_64.NC_PLC_SIGNAL_56 )
   END_RUNG
   // the same network as SCL:
   "DB2420_CNC_PLC_SIGNALS".NC_PLC_SIGNALS_33_64.NC_PLC_SIGNAL_49 := "M_ONE" AND "DB2420_CNC_PLC_SIGNALS".NC_PLC_SIGNALS_33_64.NC_PLC_SIGNAL_49;
   "DB2420_CNC_PLC_SIGNALS".NC_PLC_SIGNALS_33_64.NC_PLC_SIGNAL_50 := "M_ONE" AND "DB2420_CNC_PLC_SIGNALS".NC_PLC_SIGNALS_33_64.NC_PLC_SIGNAL_50;
   "DB2420_CNC_PLC_SIGNALS".NC_PLC_SIGNALS_33_64.NC_PLC_SIGNAL_51 := "M_ONE" AND "DB2420_CNC_PLC_SIGNALS".NC_PLC_SIGNALS_33_64.NC_PLC_SIGNAL_51;
   "DB2420_CNC_PLC_SIGNALS".NC_PLC_SIGNALS_33_64.NC_PLC_SIGNAL_52 := "M_ONE" AND "DB2420_CNC_PLC_SIGNALS".NC_PLC_SIGNALS_33_64.NC_PLC_SIGNAL_52;
   "DB2420_CNC_PLC_SIGNALS".NC_PLC_SIGNALS_33_64.NC_PLC_SIGNAL_53 := "M_ONE" AND "DB2420_CNC_PLC_SIGNALS".NC_PLC_SIGNALS_33_64.NC_PLC_SIGNAL_53;
   "DB2420_CNC_PLC_SIGNALS".NC_PLC_SIGNALS_33_64.NC_PLC_SIGNAL_54 := "M_ONE" AND "DB2420_CNC_PLC_SIGNALS".NC_PLC_SIGNALS_33_64.NC_PLC_SIGNAL_54;
   "DB2420_CNC_PLC_SIGNALS".NC_PLC_SIGNALS_33_64.NC_PLC_SIGNAL_55 := "M_ONE" AND "DB2420_CNC_PLC_SIGNALS".NC_PLC_SIGNALS_33_64.NC_PLC_SIGNAL_55;
   "DB2420_CNC_PLC_SIGNALS".NC_PLC_SIGNALS_33_64.NC_PLC_SIGNAL_56 := "M_ONE" AND "DB2420_CNC_PLC_SIGNALS".NC_PLC_SIGNALS_33_64.NC_PLC_SIGNAL_56;
END_REGION

REGION Network 12: NC PLC SIGNALS 57-64
   // SIGNAL 57 -->   FIXTURE 2 CYLINDER 9 CLAMPED
   // SIGNAL 58 -->   FIXTURE 2 CYLINDER 10 CLAMPED
   // SIGNAL 59 -->   FIXTURE 2 CYLINDER 11 CLAMPED
   // SIGNAL 60 -->   FIXTURE 2 CYLINDER 12 CLAMPED
   // SIGNAL 61 -->   FIXTURE 2 CYLINDER 13 CLAMPED
   // SIGNAL 62 -->   FIXTURE 2 CYLINDER 14 CLAMPED
   // SIGNAL 63 -->   FIXTURE 2 CYLINDER 15 CLAMPED
   // SIGNAL 64 -->   FIXTURE 2 CYLINDER 16 CLAMPED
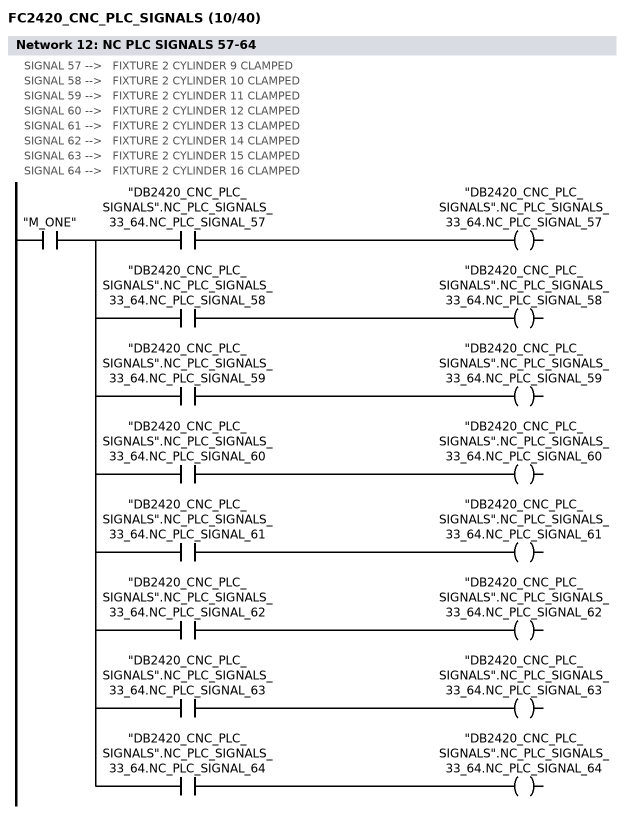
   RUNG wire#powerrail
      Contact( "M_ONE" )
      wire#w1
      Contact( "DB2420_CNC_PLC_SIGNALS".NC_PLC_SIGNALS_33_64.NC_PLC_SIGNAL_57 )
      Coil( "DB2420_CNC_PLC_SIGNALS".NC_PLC_SIGNALS_33_64.NC_PLC_SIGNAL_57 )
   END_RUNG
   RUNG wire#w1
      Contact( "DB2420_CNC_PLC_SIGNALS".NC_PLC_SIGNALS_33_64.NC_PLC_SIGNAL_58 )
      Coil( "DB2420_CNC_PLC_SIGNALS".NC_PLC_SIGNALS_33_64.NC_PLC_SIGNAL_58 )
   END_RUNG
   RUNG wire#w1
      Contact( "DB2420_CNC_PLC_SIGNALS".NC_PLC_SIGNALS_33_64.NC_PLC_SIGNAL_59 )
      Coil( "DB2420_CNC_PLC_SIGNALS".NC_PLC_SIGNALS_33_64.NC_PLC_SIGNAL_59 )
   END_RUNG
   RUNG wire#w1
      Contact( "DB2420_CNC_PLC_SIGNALS".NC_PLC_SIGNALS_33_64.NC_PLC_SIGNAL_60 )
      Coil( "DB2420_CNC_PLC_SIGNALS".NC_PLC_SIGNALS_33_64.NC_PLC_SIGNAL_60 )
   END_RUNG
   RUNG wire#w1
      Contact( "DB2420_CNC_PLC_SIGNALS".NC_PLC_SIGNALS_33_64.NC_PLC_SIGNAL_61 )
      Coil( "DB2420_CNC_PLC_SIGNALS".NC_PLC_SIGNALS_33_64.NC_PLC_SIGNAL_61 )
   END_RUNG
   RUNG wire#w1
      Contact( "DB2420_CNC_PLC_SIGNALS".NC_PLC_SIGNALS_33_64.NC_PLC_SIGNAL_62 )
      Coil( "DB2420_CNC_PLC_SIGNALS".NC_PLC_SIGNALS_33_64.NC_PLC_SIGNAL_62 )
   END_RUNG
   RUNG wire#w1
      Contact( "DB2420_CNC_PLC_SIGNALS".NC_PLC_SIGNALS_33_64.NC_PLC_SIGNAL_63 )
      Coil( "DB2420_CNC_PLC_SIGNALS".NC_PLC_SIGNALS_33_64.NC_PLC_SIGNAL_63 )
   END_RUNG
   RUNG wire#w1
      Contact( "DB2420_CNC_PLC_SIGNALS".NC_PLC_SIGNALS_33_64.NC_PLC_SIGNAL_64 )
      Coil( "DB2420_CNC_PLC_SIGNALS".NC_PLC_SIGNALS_33_64.NC_PLC_SIGNAL_64 )
   END_RUNG
   // the same network as SCL:
   "DB2420_CNC_PLC_SIGNALS".NC_PLC_SIGNALS_33_64.NC_PLC_SIGNAL_57 := "M_ONE" AND "DB2420_CNC_PLC_SIGNALS".NC_PLC_SIGNALS_33_64.NC_PLC_SIGNAL_57;
   "DB2420_CNC_PLC_SIGNALS".NC_PLC_SIGNALS_33_64.NC_PLC_SIGNAL_58 := "M_ONE" AND "DB2420_CNC_PLC_SIGNALS".NC_PLC_SIGNALS_33_64.NC_PLC_SIGNAL_58;
   "DB2420_CNC_PLC_SIGNALS".NC_PLC_SIGNALS_33_64.NC_PLC_SIGNAL_59 := "M_ONE" AND "DB2420_CNC_PLC_SIGNALS".NC_PLC_SIGNALS_33_64.NC_PLC_SIGNAL_59;
   "DB2420_CNC_PLC_SIGNALS".NC_PLC_SIGNALS_33_64.NC_PLC_SIGNAL_60 := "M_ONE" AND "DB2420_CNC_PLC_SIGNALS".NC_PLC_SIGNALS_33_64.NC_PLC_SIGNAL_60;
   "DB2420_CNC_PLC_SIGNALS".NC_PLC_SIGNALS_33_64.NC_PLC_SIGNAL_61 := "M_ONE" AND "DB2420_CNC_PLC_SIGNALS".NC_PLC_SIGNALS_33_64.NC_PLC_SIGNAL_61;
   "DB2420_CNC_PLC_SIGNALS".NC_PLC_SIGNALS_33_64.NC_PLC_SIGNAL_62 := "M_ONE" AND "DB2420_CNC_PLC_SIGNALS".NC_PLC_SIGNALS_33_64.NC_PLC_SIGNAL_62;
   "DB2420_CNC_PLC_SIGNALS".NC_PLC_SIGNALS_33_64.NC_PLC_SIGNAL_63 := "M_ONE" AND "DB2420_CNC_PLC_SIGNALS".NC_PLC_SIGNALS_33_64.NC_PLC_SIGNAL_63;
   "DB2420_CNC_PLC_SIGNALS".NC_PLC_SIGNALS_33_64.NC_PLC_SIGNAL_64 := "M_ONE" AND "DB2420_CNC_PLC_SIGNALS".NC_PLC_SIGNALS_33_64.NC_PLC_SIGNAL_64;
END_REGION

REGION Network 13: CALL FC21 NC PLC SIGNALS- $A_DBD[4048] / WRITE UNIT CYCLE SELECTION TO CNC
   // $A_DBD[1000] IN CNC
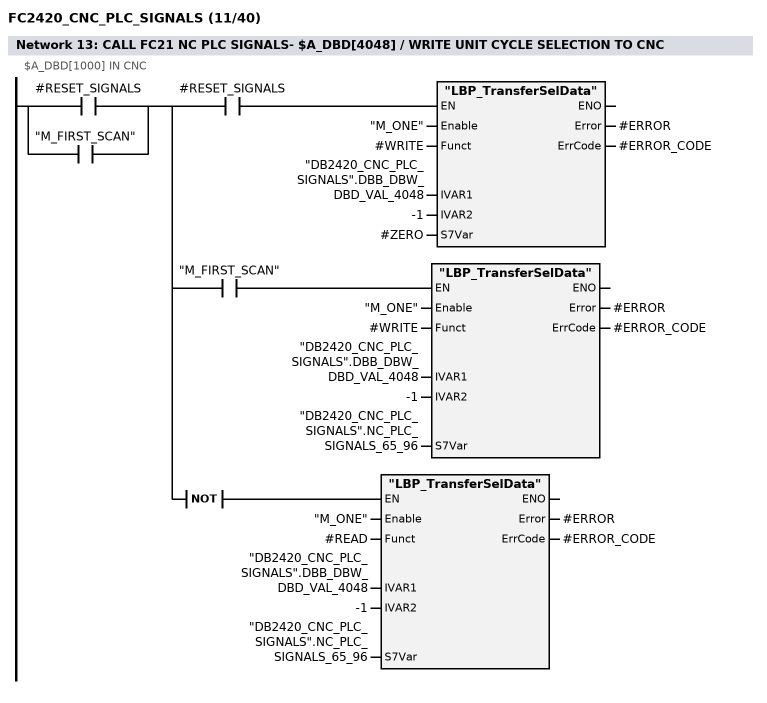
   RUNG wire#powerrail
      Contact( #RESET_SIGNALS )
      wire#w1
      Contact( #RESET_SIGNALS )
      "LBP_TransferSelData"(Enable := "M_ONE", Funct := #WRITE, IVAR1 := "DB2420_CNC_PLC_SIGNALS".DBB_DBW_DBD_VAL_4048, IVAR2 := -1, S7Var := #ZERO, Error => #ERROR, ErrCode => #ERROR_CODE)
   END_RUNG
   RUNG wire#powerrail
      Contact( "M_FIRST_SCAN" )
   END_RUNG wire#w1
   RUNG wire#w1
      Contact( "M_FIRST_SCAN" )
      "LBP_TransferSelData"(Enable := "M_ONE", Funct := #WRITE, IVAR1 := "DB2420_CNC_PLC_SIGNALS".DBB_DBW_DBD_VAL_4048, IVAR2 := -1, S7Var := "DB2420_CNC_PLC_SIGNALS".NC_PLC_SIGNALS_65_96, Error => #ERROR, ErrCode => #ERROR_CODE)
   END_RUNG
   RUNG wire#w1
      Not()
      "LBP_TransferSelData"(Enable := "M_ONE", Funct := #READ, IVAR1 := "DB2420_CNC_PLC_SIGNALS".DBB_DBW_DBD_VAL_4048, IVAR2 := -1, S7Var := "DB2420_CNC_PLC_SIGNALS".NC_PLC_SIGNALS_65_96, Error => #ERROR, ErrCode => #ERROR_CODE)
   END_RUNG
   // the same network as SCL:
   #_w1 := #RESET_SIGNALS OR "M_FIRST_SCAN";
   IF #_w1 AND #RESET_SIGNALS THEN
       "LBP_TransferSelData"(Enable := "M_ONE",
                             Funct := #WRITE,
                             IVAR1 := "DB2420_CNC_PLC_SIGNALS".DBB_DBW_DBD_VAL_4048,
                             IVAR2 := -1,
                             S7Var := #ZERO,
                             Error => #ERROR,
                             ErrCode => #ERROR_CODE);
   END_IF;
   IF #_w1 AND "M_FIRST_SCAN" THEN
       "LBP_TransferSelData"(Enable := "M_ONE",
                             Funct := #WRITE,
                             IVAR1 := "DB2420_CNC_PLC_SIGNALS".DBB_DBW_DBD_VAL_4048,
                             IVAR2 := -1,
                             S7Var := "DB2420_CNC_PLC_SIGNALS".NC_PLC_SIGNALS_65_96,
                             Error => #ERROR,
                             ErrCode => #ERROR_CODE);
   END_IF;
   IF NOT #_w1 THEN
       "LBP_TransferSelData"(Enable := "M_ONE",
                             Funct := #READ,
                             IVAR1 := "DB2420_CNC_PLC_SIGNALS".DBB_DBW_DBD_VAL_4048,
                             IVAR2 := -1,
                             S7Var := "DB2420_CNC_PLC_SIGNALS".NC_PLC_SIGNALS_65_96,
                             Error => #ERROR,
                             ErrCode => #ERROR_CODE);
   END_IF;
END_REGION

REGION Network 14: NC PLC SIGNALS 65-72
   // SIGNAL 65 -->   FIXTURE 2 CYLINDER 17 CLAMPED
   // SIGNAL 66 -->   FIXTURE 2 CYLINDER 18 CLAMPED
   // SIGNAL 67 -->   FIXTURE 2 CYLINDER 19 CLAMPED
   // SIGNAL 68 -->   FIXTURE 2 CYLINDER 20 CLAMPED
   // SIGNAL 69 -->   FIXTURE 2 CYLINDER 21 CLAMPED
   // SIGNAL 70 -->   FIXTURE 2 CYLINDER 22 CLAMPED
   // SIGNAL 71 -->   FIXTURE 2 CYLINDER 23 CLAMPED
   // SIGNAL 72 -->   FIXTURE 2 CYLINDER 24 CLAMPED
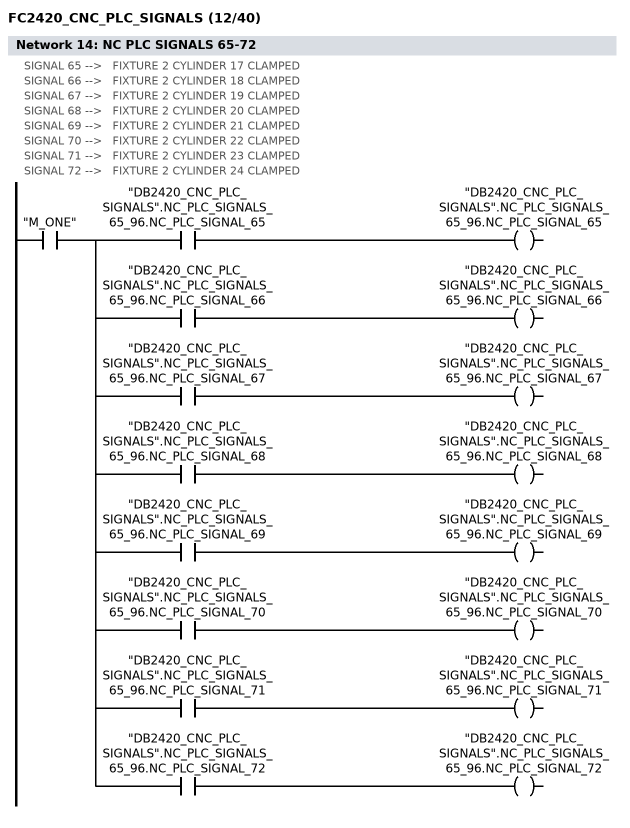
   RUNG wire#powerrail
      Contact( "M_ONE" )
      wire#w1
      Contact( "DB2420_CNC_PLC_SIGNALS".NC_PLC_SIGNALS_65_96.NC_PLC_SIGNAL_65 )
      Coil( "DB2420_CNC_PLC_SIGNALS".NC_PLC_SIGNALS_65_96.NC_PLC_SIGNAL_65 )
   END_RUNG
   RUNG wire#w1
      Contact( "DB2420_CNC_PLC_SIGNALS".NC_PLC_SIGNALS_65_96.NC_PLC_SIGNAL_66 )
      Coil( "DB2420_CNC_PLC_SIGNALS".NC_PLC_SIGNALS_65_96.NC_PLC_SIGNAL_66 )
   END_RUNG
   RUNG wire#w1
      Contact( "DB2420_CNC_PLC_SIGNALS".NC_PLC_SIGNALS_65_96.NC_PLC_SIGNAL_67 )
      Coil( "DB2420_CNC_PLC_SIGNALS".NC_PLC_SIGNALS_65_96.NC_PLC_SIGNAL_67 )
   END_RUNG
   RUNG wire#w1
      Contact( "DB2420_CNC_PLC_SIGNALS".NC_PLC_SIGNALS_65_96.NC_PLC_SIGNAL_68 )
      Coil( "DB2420_CNC_PLC_SIGNALS".NC_PLC_SIGNALS_65_96.NC_PLC_SIGNAL_68 )
   END_RUNG
   RUNG wire#w1
      Contact( "DB2420_CNC_PLC_SIGNALS".NC_PLC_SIGNALS_65_96.NC_PLC_SIGNAL_69 )
      Coil( "DB2420_CNC_PLC_SIGNALS".NC_PLC_SIGNALS_65_96.NC_PLC_SIGNAL_69 )
   END_RUNG
   RUNG wire#w1
      Contact( "DB2420_CNC_PLC_SIGNALS".NC_PLC_SIGNALS_65_96.NC_PLC_SIGNAL_70 )
      Coil( "DB2420_CNC_PLC_SIGNALS".NC_PLC_SIGNALS_65_96.NC_PLC_SIGNAL_70 )
   END_RUNG
   RUNG wire#w1
      Contact( "DB2420_CNC_PLC_SIGNALS".NC_PLC_SIGNALS_65_96.NC_PLC_SIGNAL_71 )
      Coil( "DB2420_CNC_PLC_SIGNALS".NC_PLC_SIGNALS_65_96.NC_PLC_SIGNAL_71 )
   END_RUNG
   RUNG wire#w1
      Contact( "DB2420_CNC_PLC_SIGNALS".NC_PLC_SIGNALS_65_96.NC_PLC_SIGNAL_72 )
      Coil( "DB2420_CNC_PLC_SIGNALS".NC_PLC_SIGNALS_65_96.NC_PLC_SIGNAL_72 )
   END_RUNG
   // the same network as SCL:
   "DB2420_CNC_PLC_SIGNALS".NC_PLC_SIGNALS_65_96.NC_PLC_SIGNAL_65 := "M_ONE" AND "DB2420_CNC_PLC_SIGNALS".NC_PLC_SIGNALS_65_96.NC_PLC_SIGNAL_65;
   "DB2420_CNC_PLC_SIGNALS".NC_PLC_SIGNALS_65_96.NC_PLC_SIGNAL_66 := "M_ONE" AND "DB2420_CNC_PLC_SIGNALS".NC_PLC_SIGNALS_65_96.NC_PLC_SIGNAL_66;
   "DB2420_CNC_PLC_SIGNALS".NC_PLC_SIGNALS_65_96.NC_PLC_SIGNAL_67 := "M_ONE" AND "DB2420_CNC_PLC_SIGNALS".NC_PLC_SIGNALS_65_96.NC_PLC_SIGNAL_67;
   "DB2420_CNC_PLC_SIGNALS".NC_PLC_SIGNALS_65_96.NC_PLC_SIGNAL_68 := "M_ONE" AND "DB2420_CNC_PLC_SIGNALS".NC_PLC_SIGNALS_65_96.NC_PLC_SIGNAL_68;
   "DB2420_CNC_PLC_SIGNALS".NC_PLC_SIGNALS_65_96.NC_PLC_SIGNAL_69 := "M_ONE" AND "DB2420_CNC_PLC_SIGNALS".NC_PLC_SIGNALS_65_96.NC_PLC_SIGNAL_69;
   "DB2420_CNC_PLC_SIGNALS".NC_PLC_SIGNALS_65_96.NC_PLC_SIGNAL_70 := "M_ONE" AND "DB2420_CNC_PLC_SIGNALS".NC_PLC_SIGNALS_65_96.NC_PLC_SIGNAL_70;
   "DB2420_CNC_PLC_SIGNALS".NC_PLC_SIGNALS_65_96.NC_PLC_SIGNAL_71 := "M_ONE" AND "DB2420_CNC_PLC_SIGNALS".NC_PLC_SIGNALS_65_96.NC_PLC_SIGNAL_71;
   "DB2420_CNC_PLC_SIGNALS".NC_PLC_SIGNALS_65_96.NC_PLC_SIGNAL_72 := "M_ONE" AND "DB2420_CNC_PLC_SIGNALS".NC_PLC_SIGNALS_65_96.NC_PLC_SIGNAL_72;
END_REGION

REGION Network 15: NC PLC SIGNALS 73-80
   // SIGNAL 73 --> FIXTURE 2 CYLINDER 1 UNCLAMPED
   // SIGNAL 74 --> FIXTURE 2 CYLINDER 2 UNCLAMPED
   // SIGNAL 75 --> FIXTURE 2 CYLINDER 3 UNCLAMPED
   // SIGNAL 76 --> FIXTURE 2 CYLINDER 4 UNCLAMPED
   // SIGNAL 77 --> FIXTURE 2 CYLINDER 5 UNCLAMPED
   // SIGNAL 78 --> FIXTURE 2 CYLINDER 6 UNCLAMPED
   // SIGNAL 79 --> FIXTURE 2 CYLINDER 7 UNCLAMPED
   // SIGNAL 80 --> FIXTURE 2 CYLINDER 8 UNCLAMPED
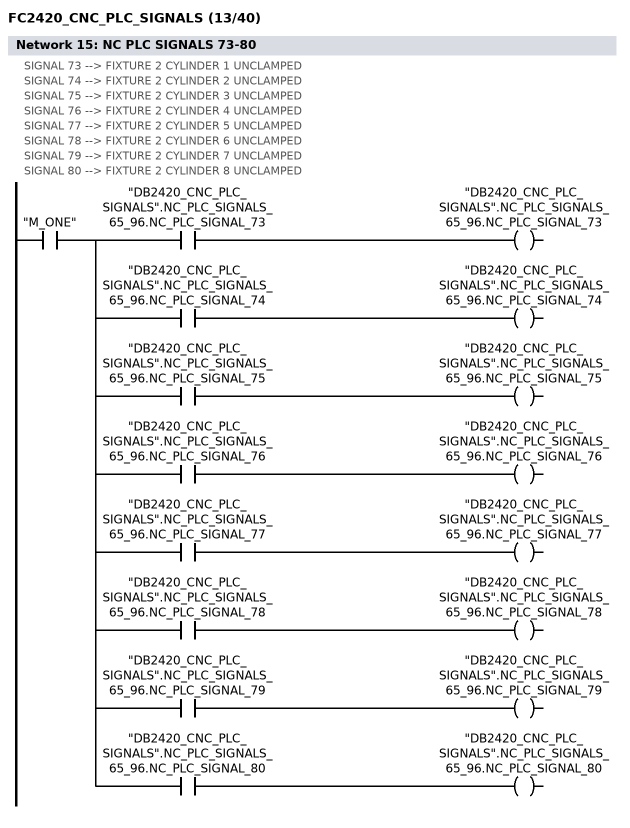
   RUNG wire#powerrail
      Contact( "M_ONE" )
      wire#w1
      Contact( "DB2420_CNC_PLC_SIGNALS".NC_PLC_SIGNALS_65_96.NC_PLC_SIGNAL_73 )
      Coil( "DB2420_CNC_PLC_SIGNALS".NC_PLC_SIGNALS_65_96.NC_PLC_SIGNAL_73 )
   END_RUNG
   RUNG wire#w1
      Contact( "DB2420_CNC_PLC_SIGNALS".NC_PLC_SIGNALS_65_96.NC_PLC_SIGNAL_74 )
      Coil( "DB2420_CNC_PLC_SIGNALS".NC_PLC_SIGNALS_65_96.NC_PLC_SIGNAL_74 )
   END_RUNG
   RUNG wire#w1
      Contact( "DB2420_CNC_PLC_SIGNALS".NC_PLC_SIGNALS_65_96.NC_PLC_SIGNAL_75 )
      Coil( "DB2420_CNC_PLC_SIGNALS".NC_PLC_SIGNALS_65_96.NC_PLC_SIGNAL_75 )
   END_RUNG
   RUNG wire#w1
      Contact( "DB2420_CNC_PLC_SIGNALS".NC_PLC_SIGNALS_65_96.NC_PLC_SIGNAL_76 )
      Coil( "DB2420_CNC_PLC_SIGNALS".NC_PLC_SIGNALS_65_96.NC_PLC_SIGNAL_76 )
   END_RUNG
   RUNG wire#w1
      Contact( "DB2420_CNC_PLC_SIGNALS".NC_PLC_SIGNALS_65_96.NC_PLC_SIGNAL_77 )
      Coil( "DB2420_CNC_PLC_SIGNALS".NC_PLC_SIGNALS_65_96.NC_PLC_SIGNAL_77 )
   END_RUNG
   RUNG wire#w1
      Contact( "DB2420_CNC_PLC_SIGNALS".NC_PLC_SIGNALS_65_96.NC_PLC_SIGNAL_78 )
      Coil( "DB2420_CNC_PLC_SIGNALS".NC_PLC_SIGNALS_65_96.NC_PLC_SIGNAL_78 )
   END_RUNG
   RUNG wire#w1
      Contact( "DB2420_CNC_PLC_SIGNALS".NC_PLC_SIGNALS_65_96.NC_PLC_SIGNAL_79 )
      Coil( "DB2420_CNC_PLC_SIGNALS".NC_PLC_SIGNALS_65_96.NC_PLC_SIGNAL_79 )
   END_RUNG
   RUNG wire#w1
      Contact( "DB2420_CNC_PLC_SIGNALS".NC_PLC_SIGNALS_65_96.NC_PLC_SIGNAL_80 )
      Coil( "DB2420_CNC_PLC_SIGNALS".NC_PLC_SIGNALS_65_96.NC_PLC_SIGNAL_80 )
   END_RUNG
   // the same network as SCL:
   "DB2420_CNC_PLC_SIGNALS".NC_PLC_SIGNALS_65_96.NC_PLC_SIGNAL_73 := "M_ONE" AND "DB2420_CNC_PLC_SIGNALS".NC_PLC_SIGNALS_65_96.NC_PLC_SIGNAL_73;
   "DB2420_CNC_PLC_SIGNALS".NC_PLC_SIGNALS_65_96.NC_PLC_SIGNAL_74 := "M_ONE" AND "DB2420_CNC_PLC_SIGNALS".NC_PLC_SIGNALS_65_96.NC_PLC_SIGNAL_74;
   "DB2420_CNC_PLC_SIGNALS".NC_PLC_SIGNALS_65_96.NC_PLC_SIGNAL_75 := "M_ONE" AND "DB2420_CNC_PLC_SIGNALS".NC_PLC_SIGNALS_65_96.NC_PLC_SIGNAL_75;
   "DB2420_CNC_PLC_SIGNALS".NC_PLC_SIGNALS_65_96.NC_PLC_SIGNAL_76 := "M_ONE" AND "DB2420_CNC_PLC_SIGNALS".NC_PLC_SIGNALS_65_96.NC_PLC_SIGNAL_76;
   "DB2420_CNC_PLC_SIGNALS".NC_PLC_SIGNALS_65_96.NC_PLC_SIGNAL_77 := "M_ONE" AND "DB2420_CNC_PLC_SIGNALS".NC_PLC_SIGNALS_65_96.NC_PLC_SIGNAL_77;
   "DB2420_CNC_PLC_SIGNALS".NC_PLC_SIGNALS_65_96.NC_PLC_SIGNAL_78 := "M_ONE" AND "DB2420_CNC_PLC_SIGNALS".NC_PLC_SIGNALS_65_96.NC_PLC_SIGNAL_78;
   "DB2420_CNC_PLC_SIGNALS".NC_PLC_SIGNALS_65_96.NC_PLC_SIGNAL_79 := "M_ONE" AND "DB2420_CNC_PLC_SIGNALS".NC_PLC_SIGNALS_65_96.NC_PLC_SIGNAL_79;
   "DB2420_CNC_PLC_SIGNALS".NC_PLC_SIGNALS_65_96.NC_PLC_SIGNAL_80 := "M_ONE" AND "DB2420_CNC_PLC_SIGNALS".NC_PLC_SIGNALS_65_96.NC_PLC_SIGNAL_80;
END_REGION

REGION Network 16: NC PLC SIGNALS 81-88
   // SIGNAL 81 --> FIXTURE 2 CYLINDER 9 UNCLAMPED
   // SIGNAL 82 --> FIXTURE 2 CYLINDER 10 UNCLAMPED
   // SIGNAL 83 --> FIXTURE 2 CYLINDER 11 UNCLAMPED
   // SIGNAL 84 --> FIXTURE 2 CYLINDER 12 UNCLAMPED
   // SIGNAL 85 --> FIXTURE 2 CYLINDER 13 UNCLAMPED
   // SIGNAL 86 --> FIXTURE 2 CYLINDER 14 UNCLAMPED
   // SIGNAL 87 --> FIXTURE 2 CYLINDER 15 UNCLAMPED
   // SIGNAL 88 --> FIXTURE 2 CYLINDER 16 UNCLAMPED
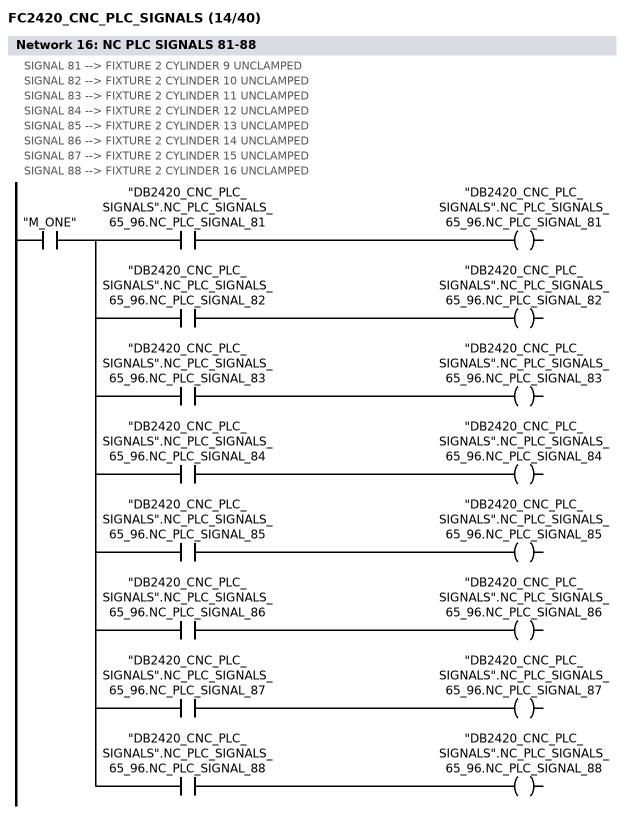
   RUNG wire#powerrail
      Contact( "M_ONE" )
      wire#w1
      Contact( "DB2420_CNC_PLC_SIGNALS".NC_PLC_SIGNALS_65_96.NC_PLC_SIGNAL_81 )
      Coil( "DB2420_CNC_PLC_SIGNALS".NC_PLC_SIGNALS_65_96.NC_PLC_SIGNAL_81 )
   END_RUNG
   RUNG wire#w1
      Contact( "DB2420_CNC_PLC_SIGNALS".NC_PLC_SIGNALS_65_96.NC_PLC_SIGNAL_82 )
      Coil( "DB2420_CNC_PLC_SIGNALS".NC_PLC_SIGNALS_65_96.NC_PLC_SIGNAL_82 )
   END_RUNG
   RUNG wire#w1
      Contact( "DB2420_CNC_PLC_SIGNALS".NC_PLC_SIGNALS_65_96.NC_PLC_SIGNAL_83 )
      Coil( "DB2420_CNC_PLC_SIGNALS".NC_PLC_SIGNALS_65_96.NC_PLC_SIGNAL_83 )
   END_RUNG
   RUNG wire#w1
      Contact( "DB2420_CNC_PLC_SIGNALS".NC_PLC_SIGNALS_65_96.NC_PLC_SIGNAL_84 )
      Coil( "DB2420_CNC_PLC_SIGNALS".NC_PLC_SIGNALS_65_96.NC_PLC_SIGNAL_84 )
   END_RUNG
   RUNG wire#w1
      Contact( "DB2420_CNC_PLC_SIGNALS".NC_PLC_SIGNALS_65_96.NC_PLC_SIGNAL_85 )
      Coil( "DB2420_CNC_PLC_SIGNALS".NC_PLC_SIGNALS_65_96.NC_PLC_SIGNAL_85 )
   END_RUNG
   RUNG wire#w1
      Contact( "DB2420_CNC_PLC_SIGNALS".NC_PLC_SIGNALS_65_96.NC_PLC_SIGNAL_86 )
      Coil( "DB2420_CNC_PLC_SIGNALS".NC_PLC_SIGNALS_65_96.NC_PLC_SIGNAL_86 )
   END_RUNG
   RUNG wire#w1
      Contact( "DB2420_CNC_PLC_SIGNALS".NC_PLC_SIGNALS_65_96.NC_PLC_SIGNAL_87 )
      Coil( "DB2420_CNC_PLC_SIGNALS".NC_PLC_SIGNALS_65_96.NC_PLC_SIGNAL_87 )
   END_RUNG
   RUNG wire#w1
      Contact( "DB2420_CNC_PLC_SIGNALS".NC_PLC_SIGNALS_65_96.NC_PLC_SIGNAL_88 )
      Coil( "DB2420_CNC_PLC_SIGNALS".NC_PLC_SIGNALS_65_96.NC_PLC_SIGNAL_88 )
   END_RUNG
   // the same network as SCL:
   "DB2420_CNC_PLC_SIGNALS".NC_PLC_SIGNALS_65_96.NC_PLC_SIGNAL_81 := "M_ONE" AND "DB2420_CNC_PLC_SIGNALS".NC_PLC_SIGNALS_65_96.NC_PLC_SIGNAL_81;
   "DB2420_CNC_PLC_SIGNALS".NC_PLC_SIGNALS_65_96.NC_PLC_SIGNAL_82 := "M_ONE" AND "DB2420_CNC_PLC_SIGNALS".NC_PLC_SIGNALS_65_96.NC_PLC_SIGNAL_82;
   "DB2420_CNC_PLC_SIGNALS".NC_PLC_SIGNALS_65_96.NC_PLC_SIGNAL_83 := "M_ONE" AND "DB2420_CNC_PLC_SIGNALS".NC_PLC_SIGNALS_65_96.NC_PLC_SIGNAL_83;
   "DB2420_CNC_PLC_SIGNALS".NC_PLC_SIGNALS_65_96.NC_PLC_SIGNAL_84 := "M_ONE" AND "DB2420_CNC_PLC_SIGNALS".NC_PLC_SIGNALS_65_96.NC_PLC_SIGNAL_84;
   "DB2420_CNC_PLC_SIGNALS".NC_PLC_SIGNALS_65_96.NC_PLC_SIGNAL_85 := "M_ONE" AND "DB2420_CNC_PLC_SIGNALS".NC_PLC_SIGNALS_65_96.NC_PLC_SIGNAL_85;
   "DB2420_CNC_PLC_SIGNALS".NC_PLC_SIGNALS_65_96.NC_PLC_SIGNAL_86 := "M_ONE" AND "DB2420_CNC_PLC_SIGNALS".NC_PLC_SIGNALS_65_96.NC_PLC_SIGNAL_86;
   "DB2420_CNC_PLC_SIGNALS".NC_PLC_SIGNALS_65_96.NC_PLC_SIGNAL_87 := "M_ONE" AND "DB2420_CNC_PLC_SIGNALS".NC_PLC_SIGNALS_65_96.NC_PLC_SIGNAL_87;
   "DB2420_CNC_PLC_SIGNALS".NC_PLC_SIGNALS_65_96.NC_PLC_SIGNAL_88 := "M_ONE" AND "DB2420_CNC_PLC_SIGNALS".NC_PLC_SIGNALS_65_96.NC_PLC_SIGNAL_88;
END_REGION

REGION Network 17: NC PLC SIGNALS 89-96
   // SIGNAL 89 --> FIXTURE 2 CYLINDER 17 UNCLAMPED
   // SIGNAL 90 --> FIXTURE 2 CYLINDER 18 UNCLAMPED
   // SIGNAL 91 --> FIXTURE 2 CYLINDER 19 UNCLAMPED
   // SIGNAL 92 --> FIXTURE 2 CYLINDER 20 UNCLAMPED
   // SIGNAL 93 --> FIXTURE 2 CYLINDER 21 UNCLAMPED
   // SIGNAL 94 --> FIXTURE 2 CYLINDER 22 UNCLAMPED
   // SIGNAL 95 --> FIXTURE 2 CYLINDER 23 UNCLAMPED
   // SIGNAL 96 --> FIXTURE 2 CYLINDER 24 UNCLAMPED
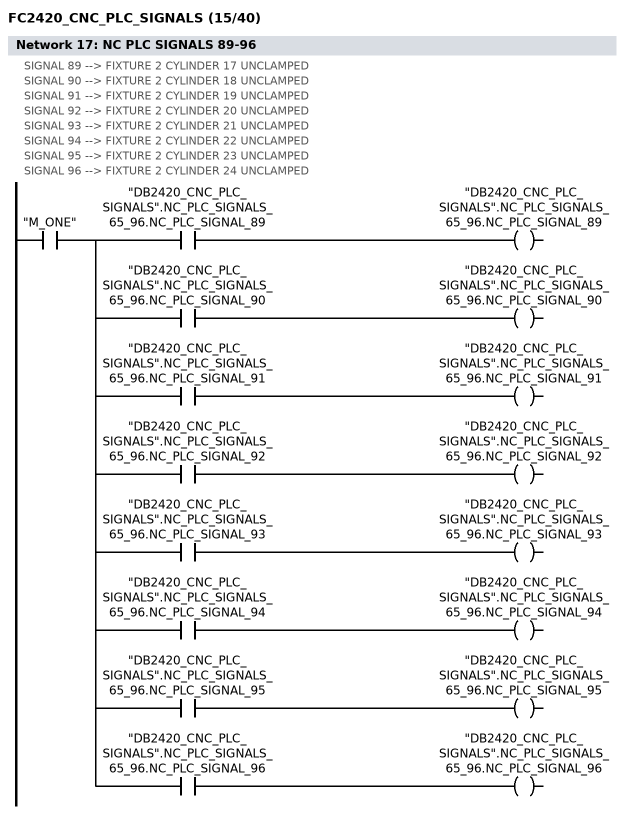
   RUNG wire#powerrail
      Contact( "M_ONE" )
      wire#w1
      Contact( "DB2420_CNC_PLC_SIGNALS".NC_PLC_SIGNALS_65_96.NC_PLC_SIGNAL_89 )
      Coil( "DB2420_CNC_PLC_SIGNALS".NC_PLC_SIGNALS_65_96.NC_PLC_SIGNAL_89 )
   END_RUNG
   RUNG wire#w1
      Contact( "DB2420_CNC_PLC_SIGNALS".NC_PLC_SIGNALS_65_96.NC_PLC_SIGNAL_90 )
      Coil( "DB2420_CNC_PLC_SIGNALS".NC_PLC_SIGNALS_65_96.NC_PLC_SIGNAL_90 )
   END_RUNG
   RUNG wire#w1
      Contact( "DB2420_CNC_PLC_SIGNALS".NC_PLC_SIGNALS_65_96.NC_PLC_SIGNAL_91 )
      Coil( "DB2420_CNC_PLC_SIGNALS".NC_PLC_SIGNALS_65_96.NC_PLC_SIGNAL_91 )
   END_RUNG
   RUNG wire#w1
      Contact( "DB2420_CNC_PLC_SIGNALS".NC_PLC_SIGNALS_65_96.NC_PLC_SIGNAL_92 )
      Coil( "DB2420_CNC_PLC_SIGNALS".NC_PLC_SIGNALS_65_96.NC_PLC_SIGNAL_92 )
   END_RUNG
   RUNG wire#w1
      Contact( "DB2420_CNC_PLC_SIGNALS".NC_PLC_SIGNALS_65_96.NC_PLC_SIGNAL_93 )
      Coil( "DB2420_CNC_PLC_SIGNALS".NC_PLC_SIGNALS_65_96.NC_PLC_SIGNAL_93 )
   END_RUNG
   RUNG wire#w1
      Contact( "DB2420_CNC_PLC_SIGNALS".NC_PLC_SIGNALS_65_96.NC_PLC_SIGNAL_94 )
      Coil( "DB2420_CNC_PLC_SIGNALS".NC_PLC_SIGNALS_65_96.NC_PLC_SIGNAL_94 )
   END_RUNG
   RUNG wire#w1
      Contact( "DB2420_CNC_PLC_SIGNALS".NC_PLC_SIGNALS_65_96.NC_PLC_SIGNAL_95 )
      Coil( "DB2420_CNC_PLC_SIGNALS".NC_PLC_SIGNALS_65_96.NC_PLC_SIGNAL_95 )
   END_RUNG
   RUNG wire#w1
      Contact( "DB2420_CNC_PLC_SIGNALS".NC_PLC_SIGNALS_65_96.NC_PLC_SIGNAL_96 )
      Coil( "DB2420_CNC_PLC_SIGNALS".NC_PLC_SIGNALS_65_96.NC_PLC_SIGNAL_96 )
   END_RUNG
   // the same network as SCL:
   "DB2420_CNC_PLC_SIGNALS".NC_PLC_SIGNALS_65_96.NC_PLC_SIGNAL_89 := "M_ONE" AND "DB2420_CNC_PLC_SIGNALS".NC_PLC_SIGNALS_65_96.NC_PLC_SIGNAL_89;
   "DB2420_CNC_PLC_SIGNALS".NC_PLC_SIGNALS_65_96.NC_PLC_SIGNAL_90 := "M_ONE" AND "DB2420_CNC_PLC_SIGNALS".NC_PLC_SIGNALS_65_96.NC_PLC_SIGNAL_90;
   "DB2420_CNC_PLC_SIGNALS".NC_PLC_SIGNALS_65_96.NC_PLC_SIGNAL_91 := "M_ONE" AND "DB2420_CNC_PLC_SIGNALS".NC_PLC_SIGNALS_65_96.NC_PLC_SIGNAL_91;
   "DB2420_CNC_PLC_SIGNALS".NC_PLC_SIGNALS_65_96.NC_PLC_SIGNAL_92 := "M_ONE" AND "DB2420_CNC_PLC_SIGNALS".NC_PLC_SIGNALS_65_96.NC_PLC_SIGNAL_92;
   "DB2420_CNC_PLC_SIGNALS".NC_PLC_SIGNALS_65_96.NC_PLC_SIGNAL_93 := "M_ONE" AND "DB2420_CNC_PLC_SIGNALS".NC_PLC_SIGNALS_65_96.NC_PLC_SIGNAL_93;
   "DB2420_CNC_PLC_SIGNALS".NC_PLC_SIGNALS_65_96.NC_PLC_SIGNAL_94 := "M_ONE" AND "DB2420_CNC_PLC_SIGNALS".NC_PLC_SIGNALS_65_96.NC_PLC_SIGNAL_94;
   "DB2420_CNC_PLC_SIGNALS".NC_PLC_SIGNALS_65_96.NC_PLC_SIGNAL_95 := "M_ONE" AND "DB2420_CNC_PLC_SIGNALS".NC_PLC_SIGNALS_65_96.NC_PLC_SIGNAL_95;
   "DB2420_CNC_PLC_SIGNALS".NC_PLC_SIGNALS_65_96.NC_PLC_SIGNAL_96 := "M_ONE" AND "DB2420_CNC_PLC_SIGNALS".NC_PLC_SIGNALS_65_96.NC_PLC_SIGNAL_96;
END_REGION

REGION Network 18: CALL FC21 NC PLC SIGNALS- $A_DBD[4052] / WRITE UNIT CYCLE SELECTION TO CNC
   // $A_DBD[1000] IN CNC
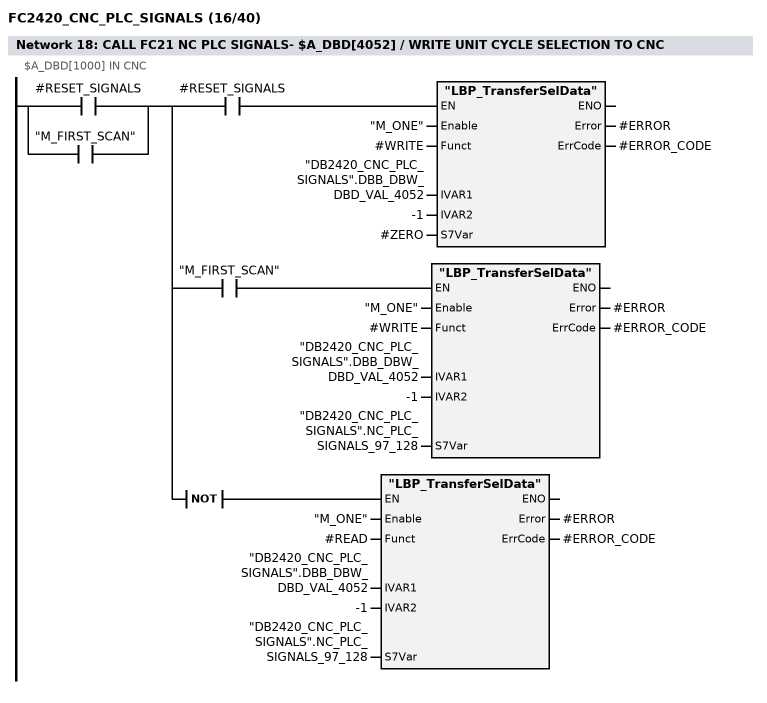
   RUNG wire#powerrail
      Contact( #RESET_SIGNALS )
      wire#w1
      Contact( #RESET_SIGNALS )
      "LBP_TransferSelData"(Enable := "M_ONE", Funct := #WRITE, IVAR1 := "DB2420_CNC_PLC_SIGNALS".DBB_DBW_DBD_VAL_4052, IVAR2 := -1, S7Var := #ZERO, Error => #ERROR, ErrCode => #ERROR_CODE)
   END_RUNG
   RUNG wire#powerrail
      Contact( "M_FIRST_SCAN" )
   END_RUNG wire#w1
   RUNG wire#w1
      Contact( "M_FIRST_SCAN" )
      "LBP_TransferSelData"(Enable := "M_ONE", Funct := #WRITE, IVAR1 := "DB2420_CNC_PLC_SIGNALS".DBB_DBW_DBD_VAL_4052, IVAR2 := -1, S7Var := "DB2420_CNC_PLC_SIGNALS".NC_PLC_SIGNALS_97_128, Error => #ERROR, ErrCode => #ERROR_CODE)
   END_RUNG
   RUNG wire#w1
      Not()
      "LBP_TransferSelData"(Enable := "M_ONE", Funct := #READ, IVAR1 := "DB2420_CNC_PLC_SIGNALS".DBB_DBW_DBD_VAL_4052, IVAR2 := -1, S7Var := "DB2420_CNC_PLC_SIGNALS".NC_PLC_SIGNALS_97_128, Error => #ERROR, ErrCode => #ERROR_CODE)
   END_RUNG
   // the same network as SCL:
   #_w1 := #RESET_SIGNALS OR "M_FIRST_SCAN";
   IF #_w1 AND #RESET_SIGNALS THEN
       "LBP_TransferSelData"(Enable := "M_ONE",
                             Funct := #WRITE,
                             IVAR1 := "DB2420_CNC_PLC_SIGNALS".DBB_DBW_DBD_VAL_4052,
                             IVAR2 := -1,
                             S7Var := #ZERO,
                             Error => #ERROR,
                             ErrCode => #ERROR_CODE);
   END_IF;
   IF #_w1 AND "M_FIRST_SCAN" THEN
       "LBP_TransferSelData"(Enable := "M_ONE",
                             Funct := #WRITE,
                             IVAR1 := "DB2420_CNC_PLC_SIGNALS".DBB_DBW_DBD_VAL_4052,
                             IVAR2 := -1,
                             S7Var := "DB2420_CNC_PLC_SIGNALS".NC_PLC_SIGNALS_97_128,
                             Error => #ERROR,
                             ErrCode => #ERROR_CODE);
   END_IF;
   IF NOT #_w1 THEN
       "LBP_TransferSelData"(Enable := "M_ONE",
                             Funct := #READ,
                             IVAR1 := "DB2420_CNC_PLC_SIGNALS".DBB_DBW_DBD_VAL_4052,
                             IVAR2 := -1,
                             S7Var := "DB2420_CNC_PLC_SIGNALS".NC_PLC_SIGNALS_97_128,
                             Error => #ERROR,
                             ErrCode => #ERROR_CODE);
   END_IF;
END_REGION

REGION Network 19: NC PLC SIGNALS 97-104
   // SIGNAL 97 --> SPARE
   // SIGNAL 98 --> SPARE
   // SIGNAL 99 --> SPARE
   // SIGNAL100 --> SPARE
   // SIGNAL 101 --> SPARE
   // SIGNAL 102 --> SPARE
   // SIGNAL 103 --> SPARE
   // SIGNAL 104 --> SPARE
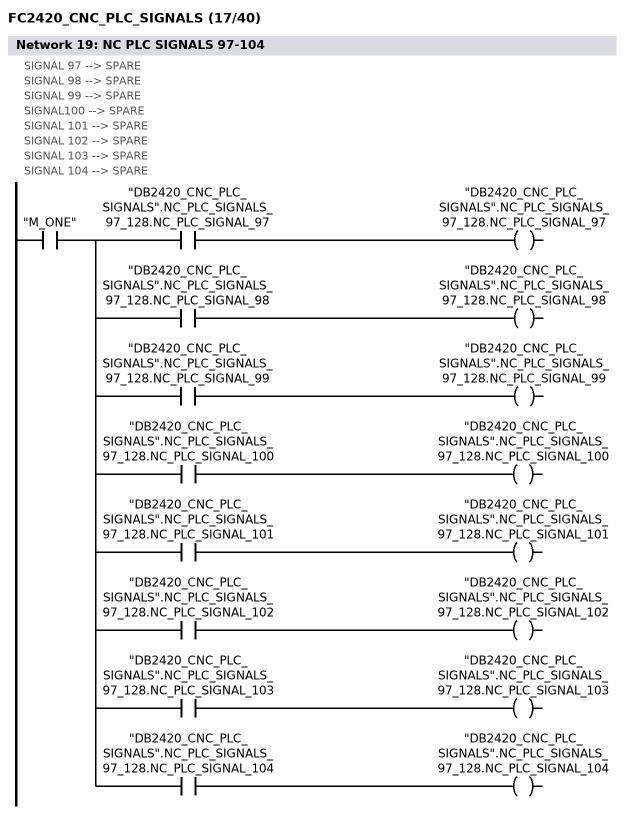
   RUNG wire#powerrail
      Contact( "M_ONE" )
      wire#w1
      Contact( "DB2420_CNC_PLC_SIGNALS".NC_PLC_SIGNALS_97_128.NC_PLC_SIGNAL_97 )
      Coil( "DB2420_CNC_PLC_SIGNALS".NC_PLC_SIGNALS_97_128.NC_PLC_SIGNAL_97 )
   END_RUNG
   RUNG wire#w1
      Contact( "DB2420_CNC_PLC_SIGNALS".NC_PLC_SIGNALS_97_128.NC_PLC_SIGNAL_98 )
      Coil( "DB2420_CNC_PLC_SIGNALS".NC_PLC_SIGNALS_97_128.NC_PLC_SIGNAL_98 )
   END_RUNG
   RUNG wire#w1
      Contact( "DB2420_CNC_PLC_SIGNALS".NC_PLC_SIGNALS_97_128.NC_PLC_SIGNAL_99 )
      Coil( "DB2420_CNC_PLC_SIGNALS".NC_PLC_SIGNALS_97_128.NC_PLC_SIGNAL_99 )
   END_RUNG
   RUNG wire#w1
      Contact( "DB2420_CNC_PLC_SIGNALS".NC_PLC_SIGNALS_97_128.NC_PLC_SIGNAL_100 )
      Coil( "DB2420_CNC_PLC_SIGNALS".NC_PLC_SIGNALS_97_128.NC_PLC_SIGNAL_100 )
   END_RUNG
   RUNG wire#w1
      Contact( "DB2420_CNC_PLC_SIGNALS".NC_PLC_SIGNALS_97_128.NC_PLC_SIGNAL_101 )
      Coil( "DB2420_CNC_PLC_SIGNALS".NC_PLC_SIGNALS_97_128.NC_PLC_SIGNAL_101 )
   END_RUNG
   RUNG wire#w1
      Contact( "DB2420_CNC_PLC_SIGNALS".NC_PLC_SIGNALS_97_128.NC_PLC_SIGNAL_102 )
      Coil( "DB2420_CNC_PLC_SIGNALS".NC_PLC_SIGNALS_97_128.NC_PLC_SIGNAL_102 )
   END_RUNG
   RUNG wire#w1
      Contact( "DB2420_CNC_PLC_SIGNALS".NC_PLC_SIGNALS_97_128.NC_PLC_SIGNAL_103 )
      Coil( "DB2420_CNC_PLC_SIGNALS".NC_PLC_SIGNALS_97_128.NC_PLC_SIGNAL_103 )
   END_RUNG
   RUNG wire#w1
      Contact( "DB2420_CNC_PLC_SIGNALS".NC_PLC_SIGNALS_97_128.NC_PLC_SIGNAL_104 )
      Coil( "DB2420_CNC_PLC_SIGNALS".NC_PLC_SIGNALS_97_128.NC_PLC_SIGNAL_104 )
   END_RUNG
   // the same network as SCL:
   "DB2420_CNC_PLC_SIGNALS".NC_PLC_SIGNALS_97_128.NC_PLC_SIGNAL_97 := "M_ONE" AND "DB2420_CNC_PLC_SIGNALS".NC_PLC_SIGNALS_97_128.NC_PLC_SIGNAL_97;
   "DB2420_CNC_PLC_SIGNALS".NC_PLC_SIGNALS_97_128.NC_PLC_SIGNAL_98 := "M_ONE" AND "DB2420_CNC_PLC_SIGNALS".NC_PLC_SIGNALS_97_128.NC_PLC_SIGNAL_98;
   "DB2420_CNC_PLC_SIGNALS".NC_PLC_SIGNALS_97_128.NC_PLC_SIGNAL_99 := "M_ONE" AND "DB2420_CNC_PLC_SIGNALS".NC_PLC_SIGNALS_97_128.NC_PLC_SIGNAL_99;
   "DB2420_CNC_PLC_SIGNALS".NC_PLC_SIGNALS_97_128.NC_PLC_SIGNAL_100 := "M_ONE" AND "DB2420_CNC_PLC_SIGNALS".NC_PLC_SIGNALS_97_128.NC_PLC_SIGNAL_100;
   "DB2420_CNC_PLC_SIGNALS".NC_PLC_SIGNALS_97_128.NC_PLC_SIGNAL_101 := "M_ONE" AND "DB2420_CNC_PLC_SIGNALS".NC_PLC_SIGNALS_97_128.NC_PLC_SIGNAL_101;
   "DB2420_CNC_PLC_SIGNALS".NC_PLC_SIGNALS_97_128.NC_PLC_SIGNAL_102 := "M_ONE" AND "DB2420_CNC_PLC_SIGNALS".NC_PLC_SIGNALS_97_128.NC_PLC_SIGNAL_102;
   "DB2420_CNC_PLC_SIGNALS".NC_PLC_SIGNALS_97_128.NC_PLC_SIGNAL_103 := "M_ONE" AND "DB2420_CNC_PLC_SIGNALS".NC_PLC_SIGNALS_97_128.NC_PLC_SIGNAL_103;
   "DB2420_CNC_PLC_SIGNALS".NC_PLC_SIGNALS_97_128.NC_PLC_SIGNAL_104 := "M_ONE" AND "DB2420_CNC_PLC_SIGNALS".NC_PLC_SIGNALS_97_128.NC_PLC_SIGNAL_104;
END_REGION

REGION Network 20: NC PLC SIGNALS 105-112
   // SIGNAL 105 --> SPARE
   // SIGNAL 106 --> SPARE
   // SIGNAL 107 --> SPARE
   // SIGNAL 108 --> SPARE
   // SIGNAL 109 --> SPARE
   // SIGNAL 110 --> SPARE
   // SIGNAL 111 --> SPARE
   // SIGNAL 112 --> SPARE
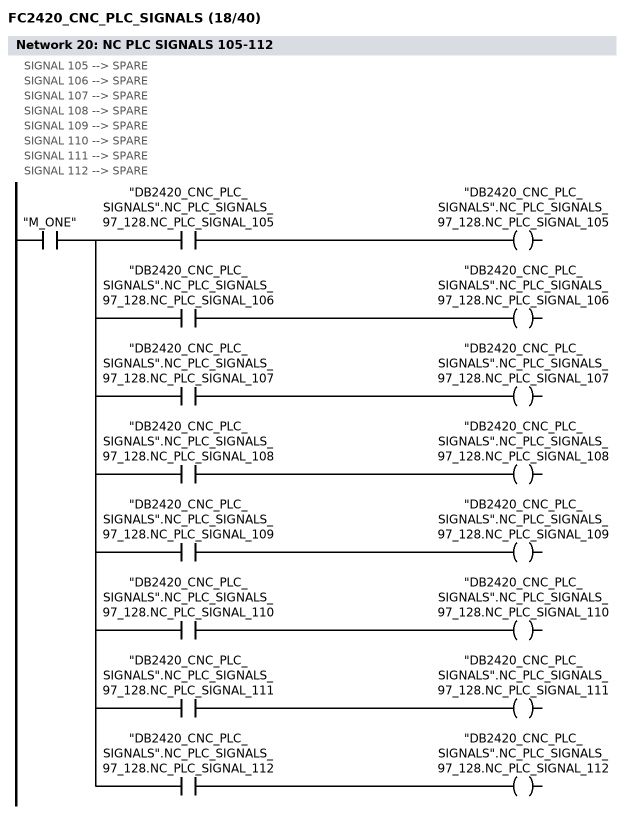
   RUNG wire#powerrail
      Contact( "M_ONE" )
      wire#w1
      Contact( "DB2420_CNC_PLC_SIGNALS".NC_PLC_SIGNALS_97_128.NC_PLC_SIGNAL_105 )
      Coil( "DB2420_CNC_PLC_SIGNALS".NC_PLC_SIGNALS_97_128.NC_PLC_SIGNAL_105 )
   END_RUNG
   RUNG wire#w1
      Contact( "DB2420_CNC_PLC_SIGNALS".NC_PLC_SIGNALS_97_128.NC_PLC_SIGNAL_106 )
      Coil( "DB2420_CNC_PLC_SIGNALS".NC_PLC_SIGNALS_97_128.NC_PLC_SIGNAL_106 )
   END_RUNG
   RUNG wire#w1
      Contact( "DB2420_CNC_PLC_SIGNALS".NC_PLC_SIGNALS_97_128.NC_PLC_SIGNAL_107 )
      Coil( "DB2420_CNC_PLC_SIGNALS".NC_PLC_SIGNALS_97_128.NC_PLC_SIGNAL_107 )
   END_RUNG
   RUNG wire#w1
      Contact( "DB2420_CNC_PLC_SIGNALS".NC_PLC_SIGNALS_97_128.NC_PLC_SIGNAL_108 )
      Coil( "DB2420_CNC_PLC_SIGNALS".NC_PLC_SIGNALS_97_128.NC_PLC_SIGNAL_108 )
   END_RUNG
   RUNG wire#w1
      Contact( "DB2420_CNC_PLC_SIGNALS".NC_PLC_SIGNALS_97_128.NC_PLC_SIGNAL_109 )
      Coil( "DB2420_CNC_PLC_SIGNALS".NC_PLC_SIGNALS_97_128.NC_PLC_SIGNAL_109 )
   END_RUNG
   RUNG wire#w1
      Contact( "DB2420_CNC_PLC_SIGNALS".NC_PLC_SIGNALS_97_128.NC_PLC_SIGNAL_110 )
      Coil( "DB2420_CNC_PLC_SIGNALS".NC_PLC_SIGNALS_97_128.NC_PLC_SIGNAL_110 )
   END_RUNG
   RUNG wire#w1
      Contact( "DB2420_CNC_PLC_SIGNALS".NC_PLC_SIGNALS_97_128.NC_PLC_SIGNAL_111 )
      Coil( "DB2420_CNC_PLC_SIGNALS".NC_PLC_SIGNALS_97_128.NC_PLC_SIGNAL_111 )
   END_RUNG
   RUNG wire#w1
      Contact( "DB2420_CNC_PLC_SIGNALS".NC_PLC_SIGNALS_97_128.NC_PLC_SIGNAL_112 )
      Coil( "DB2420_CNC_PLC_SIGNALS".NC_PLC_SIGNALS_97_128.NC_PLC_SIGNAL_112 )
   END_RUNG
   // the same network as SCL:
   "DB2420_CNC_PLC_SIGNALS".NC_PLC_SIGNALS_97_128.NC_PLC_SIGNAL_105 := "M_ONE" AND "DB2420_CNC_PLC_SIGNALS".NC_PLC_SIGNALS_97_128.NC_PLC_SIGNAL_105;
   "DB2420_CNC_PLC_SIGNALS".NC_PLC_SIGNALS_97_128.NC_PLC_SIGNAL_106 := "M_ONE" AND "DB2420_CNC_PLC_SIGNALS".NC_PLC_SIGNALS_97_128.NC_PLC_SIGNAL_106;
   "DB2420_CNC_PLC_SIGNALS".NC_PLC_SIGNALS_97_128.NC_PLC_SIGNAL_107 := "M_ONE" AND "DB2420_CNC_PLC_SIGNALS".NC_PLC_SIGNALS_97_128.NC_PLC_SIGNAL_107;
   "DB2420_CNC_PLC_SIGNALS".NC_PLC_SIGNALS_97_128.NC_PLC_SIGNAL_108 := "M_ONE" AND "DB2420_CNC_PLC_SIGNALS".NC_PLC_SIGNALS_97_128.NC_PLC_SIGNAL_108;
   "DB2420_CNC_PLC_SIGNALS".NC_PLC_SIGNALS_97_128.NC_PLC_SIGNAL_109 := "M_ONE" AND "DB2420_CNC_PLC_SIGNALS".NC_PLC_SIGNALS_97_128.NC_PLC_SIGNAL_109;
   "DB2420_CNC_PLC_SIGNALS".NC_PLC_SIGNALS_97_128.NC_PLC_SIGNAL_110 := "M_ONE" AND "DB2420_CNC_PLC_SIGNALS".NC_PLC_SIGNALS_97_128.NC_PLC_SIGNAL_110;
   "DB2420_CNC_PLC_SIGNALS".NC_PLC_SIGNALS_97_128.NC_PLC_SIGNAL_111 := "M_ONE" AND "DB2420_CNC_PLC_SIGNALS".NC_PLC_SIGNALS_97_128.NC_PLC_SIGNAL_111;
   "DB2420_CNC_PLC_SIGNALS".NC_PLC_SIGNALS_97_128.NC_PLC_SIGNAL_112 := "M_ONE" AND "DB2420_CNC_PLC_SIGNALS".NC_PLC_SIGNALS_97_128.NC_PLC_SIGNAL_112;
END_REGION

REGION Network 21: NC PLC SIGNALS 113-120
   // SIGNAL 113 --> SPARE
   // SIGNAL 114 --> SPARE
   // SIGNAL 115 --> SPARE
   // SIGNAL 116 --> SPARE
   // SIGNAL 117 --> SPARE
   // SIGNAL 118 --> SPARE
   // SIGNAL 119 --> SPARE
   // SIGNAL 120 --> SPARE
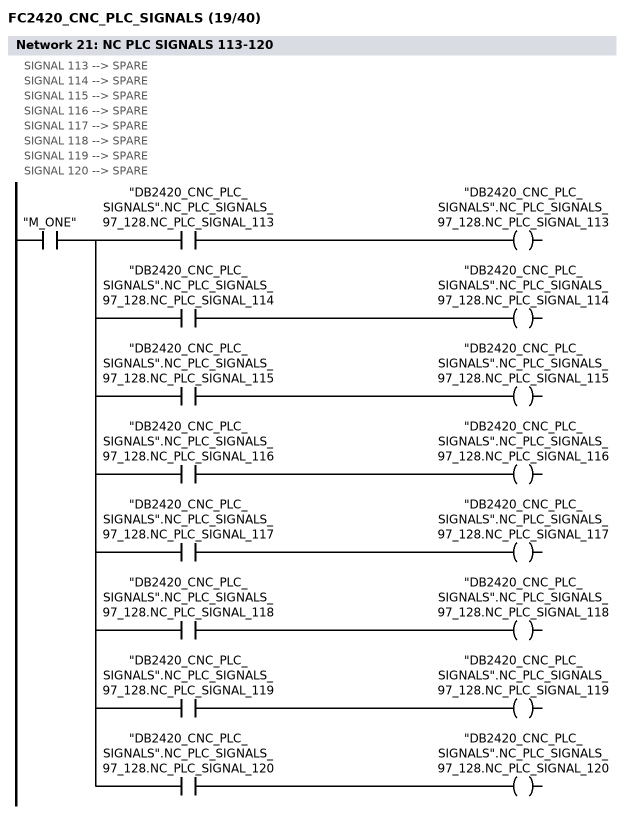
   RUNG wire#powerrail
      Contact( "M_ONE" )
      wire#w1
      Contact( "DB2420_CNC_PLC_SIGNALS".NC_PLC_SIGNALS_97_128.NC_PLC_SIGNAL_113 )
      Coil( "DB2420_CNC_PLC_SIGNALS".NC_PLC_SIGNALS_97_128.NC_PLC_SIGNAL_113 )
   END_RUNG
   RUNG wire#w1
      Contact( "DB2420_CNC_PLC_SIGNALS".NC_PLC_SIGNALS_97_128.NC_PLC_SIGNAL_114 )
      Coil( "DB2420_CNC_PLC_SIGNALS".NC_PLC_SIGNALS_97_128.NC_PLC_SIGNAL_114 )
   END_RUNG
   RUNG wire#w1
      Contact( "DB2420_CNC_PLC_SIGNALS".NC_PLC_SIGNALS_97_128.NC_PLC_SIGNAL_115 )
      Coil( "DB2420_CNC_PLC_SIGNALS".NC_PLC_SIGNALS_97_128.NC_PLC_SIGNAL_115 )
   END_RUNG
   RUNG wire#w1
      Contact( "DB2420_CNC_PLC_SIGNALS".NC_PLC_SIGNALS_97_128.NC_PLC_SIGNAL_116 )
      Coil( "DB2420_CNC_PLC_SIGNALS".NC_PLC_SIGNALS_97_128.NC_PLC_SIGNAL_116 )
   END_RUNG
   RUNG wire#w1
      Contact( "DB2420_CNC_PLC_SIGNALS".NC_PLC_SIGNALS_97_128.NC_PLC_SIGNAL_117 )
      Coil( "DB2420_CNC_PLC_SIGNALS".NC_PLC_SIGNALS_97_128.NC_PLC_SIGNAL_117 )
   END_RUNG
   RUNG wire#w1
      Contact( "DB2420_CNC_PLC_SIGNALS".NC_PLC_SIGNALS_97_128.NC_PLC_SIGNAL_118 )
      Coil( "DB2420_CNC_PLC_SIGNALS".NC_PLC_SIGNALS_97_128.NC_PLC_SIGNAL_118 )
   END_RUNG
   RUNG wire#w1
      Contact( "DB2420_CNC_PLC_SIGNALS".NC_PLC_SIGNALS_97_128.NC_PLC_SIGNAL_119 )
      Coil( "DB2420_CNC_PLC_SIGNALS".NC_PLC_SIGNALS_97_128.NC_PLC_SIGNAL_119 )
   END_RUNG
   RUNG wire#w1
      Contact( "DB2420_CNC_PLC_SIGNALS".NC_PLC_SIGNALS_97_128.NC_PLC_SIGNAL_120 )
      Coil( "DB2420_CNC_PLC_SIGNALS".NC_PLC_SIGNALS_97_128.NC_PLC_SIGNAL_120 )
   END_RUNG
   // the same network as SCL:
   "DB2420_CNC_PLC_SIGNALS".NC_PLC_SIGNALS_97_128.NC_PLC_SIGNAL_113 := "M_ONE" AND "DB2420_CNC_PLC_SIGNALS".NC_PLC_SIGNALS_97_128.NC_PLC_SIGNAL_113;
   "DB2420_CNC_PLC_SIGNALS".NC_PLC_SIGNALS_97_128.NC_PLC_SIGNAL_114 := "M_ONE" AND "DB2420_CNC_PLC_SIGNALS".NC_PLC_SIGNALS_97_128.NC_PLC_SIGNAL_114;
   "DB2420_CNC_PLC_SIGNALS".NC_PLC_SIGNALS_97_128.NC_PLC_SIGNAL_115 := "M_ONE" AND "DB2420_CNC_PLC_SIGNALS".NC_PLC_SIGNALS_97_128.NC_PLC_SIGNAL_115;
   "DB2420_CNC_PLC_SIGNALS".NC_PLC_SIGNALS_97_128.NC_PLC_SIGNAL_116 := "M_ONE" AND "DB2420_CNC_PLC_SIGNALS".NC_PLC_SIGNALS_97_128.NC_PLC_SIGNAL_116;
   "DB2420_CNC_PLC_SIGNALS".NC_PLC_SIGNALS_97_128.NC_PLC_SIGNAL_117 := "M_ONE" AND "DB2420_CNC_PLC_SIGNALS".NC_PLC_SIGNALS_97_128.NC_PLC_SIGNAL_117;
   "DB2420_CNC_PLC_SIGNALS".NC_PLC_SIGNALS_97_128.NC_PLC_SIGNAL_118 := "M_ONE" AND "DB2420_CNC_PLC_SIGNALS".NC_PLC_SIGNALS_97_128.NC_PLC_SIGNAL_118;
   "DB2420_CNC_PLC_SIGNALS".NC_PLC_SIGNALS_97_128.NC_PLC_SIGNAL_119 := "M_ONE" AND "DB2420_CNC_PLC_SIGNALS".NC_PLC_SIGNALS_97_128.NC_PLC_SIGNAL_119;
   "DB2420_CNC_PLC_SIGNALS".NC_PLC_SIGNALS_97_128.NC_PLC_SIGNAL_120 := "M_ONE" AND "DB2420_CNC_PLC_SIGNALS".NC_PLC_SIGNALS_97_128.NC_PLC_SIGNAL_120;
END_REGION

REGION Network 22: NC PLC SIGNALS 121-128
   // SIGNAL 121 --> SPARE
   // SIGNAL 122 --> SPARE
   // SIGNAL 123 --> SPARE
   // SIGNAL 124 --> SPARE
   // SIGNAL 125 --> SPARE
   // SIGNAL 126 --> SPARE
   // SIGNAL 127 --> SPARE
   // SIGNAL 128 --> SPARE
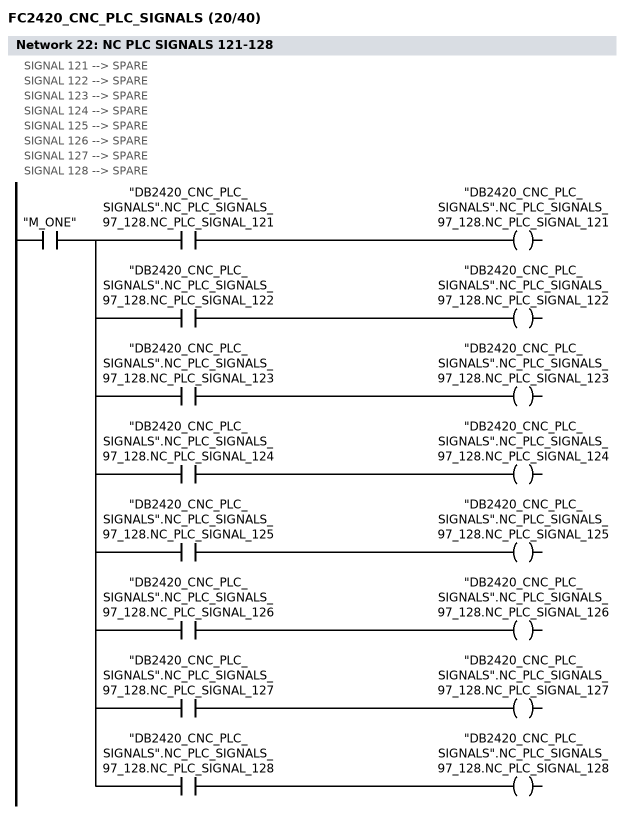
   RUNG wire#powerrail
      Contact( "M_ONE" )
      wire#w1
      Contact( "DB2420_CNC_PLC_SIGNALS".NC_PLC_SIGNALS_97_128.NC_PLC_SIGNAL_121 )
      Coil( "DB2420_CNC_PLC_SIGNALS".NC_PLC_SIGNALS_97_128.NC_PLC_SIGNAL_121 )
   END_RUNG
   RUNG wire#w1
      Contact( "DB2420_CNC_PLC_SIGNALS".NC_PLC_SIGNALS_97_128.NC_PLC_SIGNAL_122 )
      Coil( "DB2420_CNC_PLC_SIGNALS".NC_PLC_SIGNALS_97_128.NC_PLC_SIGNAL_122 )
   END_RUNG
   RUNG wire#w1
      Contact( "DB2420_CNC_PLC_SIGNALS".NC_PLC_SIGNALS_97_128.NC_PLC_SIGNAL_123 )
      Coil( "DB2420_CNC_PLC_SIGNALS".NC_PLC_SIGNALS_97_128.NC_PLC_SIGNAL_123 )
   END_RUNG
   RUNG wire#w1
      Contact( "DB2420_CNC_PLC_SIGNALS".NC_PLC_SIGNALS_97_128.NC_PLC_SIGNAL_124 )
      Coil( "DB2420_CNC_PLC_SIGNALS".NC_PLC_SIGNALS_97_128.NC_PLC_SIGNAL_124 )
   END_RUNG
   RUNG wire#w1
      Contact( "DB2420_CNC_PLC_SIGNALS".NC_PLC_SIGNALS_97_128.NC_PLC_SIGNAL_125 )
      Coil( "DB2420_CNC_PLC_SIGNALS".NC_PLC_SIGNALS_97_128.NC_PLC_SIGNAL_125 )
   END_RUNG
   RUNG wire#w1
      Contact( "DB2420_CNC_PLC_SIGNALS".NC_PLC_SIGNALS_97_128.NC_PLC_SIGNAL_126 )
      Coil( "DB2420_CNC_PLC_SIGNALS".NC_PLC_SIGNALS_97_128.NC_PLC_SIGNAL_126 )
   END_RUNG
   RUNG wire#w1
      Contact( "DB2420_CNC_PLC_SIGNALS".NC_PLC_SIGNALS_97_128.NC_PLC_SIGNAL_127 )
      Coil( "DB2420_CNC_PLC_SIGNALS".NC_PLC_SIGNALS_97_128.NC_PLC_SIGNAL_127 )
   END_RUNG
   RUNG wire#w1
      Contact( "DB2420_CNC_PLC_SIGNALS".NC_PLC_SIGNALS_97_128.NC_PLC_SIGNAL_128 )
      Coil( "DB2420_CNC_PLC_SIGNALS".NC_PLC_SIGNALS_97_128.NC_PLC_SIGNAL_128 )
   END_RUNG
   // the same network as SCL:
   "DB2420_CNC_PLC_SIGNALS".NC_PLC_SIGNALS_97_128.NC_PLC_SIGNAL_121 := "M_ONE" AND "DB2420_CNC_PLC_SIGNALS".NC_PLC_SIGNALS_97_128.NC_PLC_SIGNAL_121;
   "DB2420_CNC_PLC_SIGNALS".NC_PLC_SIGNALS_97_128.NC_PLC_SIGNAL_122 := "M_ONE" AND "DB2420_CNC_PLC_SIGNALS".NC_PLC_SIGNALS_97_128.NC_PLC_SIGNAL_122;
   "DB2420_CNC_PLC_SIGNALS".NC_PLC_SIGNALS_97_128.NC_PLC_SIGNAL_123 := "M_ONE" AND "DB2420_CNC_PLC_SIGNALS".NC_PLC_SIGNALS_97_128.NC_PLC_SIGNAL_123;
   "DB2420_CNC_PLC_SIGNALS".NC_PLC_SIGNALS_97_128.NC_PLC_SIGNAL_124 := "M_ONE" AND "DB2420_CNC_PLC_SIGNALS".NC_PLC_SIGNALS_97_128.NC_PLC_SIGNAL_124;
   "DB2420_CNC_PLC_SIGNALS".NC_PLC_SIGNALS_97_128.NC_PLC_SIGNAL_125 := "M_ONE" AND "DB2420_CNC_PLC_SIGNALS".NC_PLC_SIGNALS_97_128.NC_PLC_SIGNAL_125;
   "DB2420_CNC_PLC_SIGNALS".NC_PLC_SIGNALS_97_128.NC_PLC_SIGNAL_126 := "M_ONE" AND "DB2420_CNC_PLC_SIGNALS".NC_PLC_SIGNALS_97_128.NC_PLC_SIGNAL_126;
   "DB2420_CNC_PLC_SIGNALS".NC_PLC_SIGNALS_97_128.NC_PLC_SIGNAL_127 := "M_ONE" AND "DB2420_CNC_PLC_SIGNALS".NC_PLC_SIGNALS_97_128.NC_PLC_SIGNAL_127;
   "DB2420_CNC_PLC_SIGNALS".NC_PLC_SIGNALS_97_128.NC_PLC_SIGNAL_128 := "M_ONE" AND "DB2420_CNC_PLC_SIGNALS".NC_PLC_SIGNALS_97_128.NC_PLC_SIGNAL_128;
END_REGION

REGION Network 23: CALL FC21 NC PLC SIGNALS- $A_DBD[4056] / WRITE UNIT CYCLE SELECTION TO CNC
   // $A_DBD[1000] IN CNC
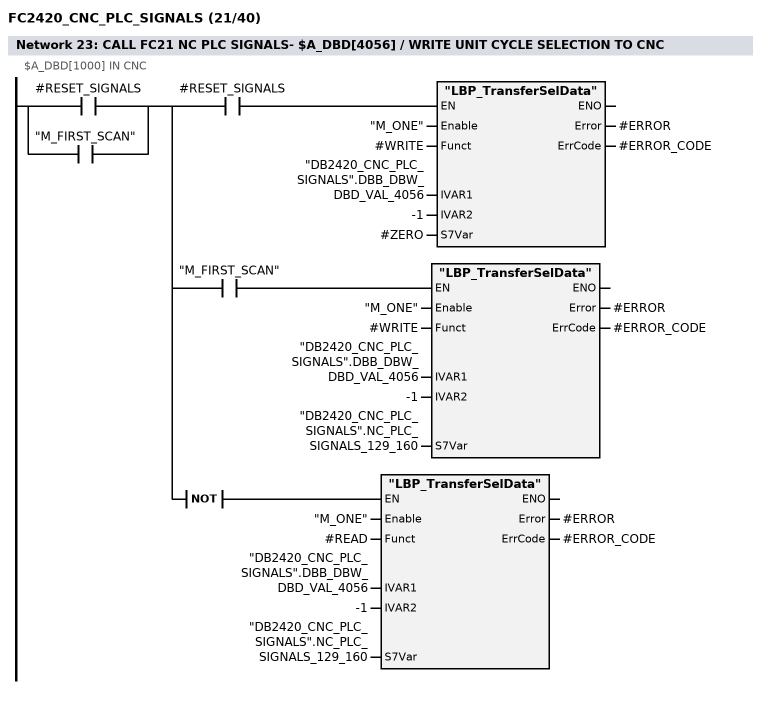
   RUNG wire#powerrail
      Contact( #RESET_SIGNALS )
      wire#w1
      Contact( #RESET_SIGNALS )
      "LBP_TransferSelData"(Enable := "M_ONE", Funct := #WRITE, IVAR1 := "DB2420_CNC_PLC_SIGNALS".DBB_DBW_DBD_VAL_4056, IVAR2 := -1, S7Var := #ZERO, Error => #ERROR, ErrCode => #ERROR_CODE)
   END_RUNG
   RUNG wire#powerrail
      Contact( "M_FIRST_SCAN" )
   END_RUNG wire#w1
   RUNG wire#w1
      Contact( "M_FIRST_SCAN" )
      "LBP_TransferSelData"(Enable := "M_ONE", Funct := #WRITE, IVAR1 := "DB2420_CNC_PLC_SIGNALS".DBB_DBW_DBD_VAL_4056, IVAR2 := -1, S7Var := "DB2420_CNC_PLC_SIGNALS".NC_PLC_SIGNALS_129_160, Error => #ERROR, ErrCode => #ERROR_CODE)
   END_RUNG
   RUNG wire#w1
      Not()
      "LBP_TransferSelData"(Enable := "M_ONE", Funct := #READ, IVAR1 := "DB2420_CNC_PLC_SIGNALS".DBB_DBW_DBD_VAL_4056, IVAR2 := -1, S7Var := "DB2420_CNC_PLC_SIGNALS".NC_PLC_SIGNALS_129_160, Error => #ERROR, ErrCode => #ERROR_CODE)
   END_RUNG
   // the same network as SCL:
   #_w1 := #RESET_SIGNALS OR "M_FIRST_SCAN";
   IF #_w1 AND #RESET_SIGNALS THEN
       "LBP_TransferSelData"(Enable := "M_ONE",
                             Funct := #WRITE,
                             IVAR1 := "DB2420_CNC_PLC_SIGNALS".DBB_DBW_DBD_VAL_4056,
                             IVAR2 := -1,
                             S7Var := #ZERO,
                             Error => #ERROR,
                             ErrCode => #ERROR_CODE);
   END_IF;
   IF #_w1 AND "M_FIRST_SCAN" THEN
       "LBP_TransferSelData"(Enable := "M_ONE",
                             Funct := #WRITE,
                             IVAR1 := "DB2420_CNC_PLC_SIGNALS".DBB_DBW_DBD_VAL_4056,
                             IVAR2 := -1,
                             S7Var := "DB2420_CNC_PLC_SIGNALS".NC_PLC_SIGNALS_129_160,
                             Error => #ERROR,
                             ErrCode => #ERROR_CODE);
   END_IF;
   IF NOT #_w1 THEN
       "LBP_TransferSelData"(Enable := "M_ONE",
                             Funct := #READ,
                             IVAR1 := "DB2420_CNC_PLC_SIGNALS".DBB_DBW_DBD_VAL_4056,
                             IVAR2 := -1,
                             S7Var := "DB2420_CNC_PLC_SIGNALS".NC_PLC_SIGNALS_129_160,
                             Error => #ERROR,
                             ErrCode => #ERROR_CODE);
   END_IF;
END_REGION

REGION Network 24: NC PLC SIGNALS 129-136
   // SIGNAL 129 --> SPARE
   // SIGNAL 130 --> SPARE
   // SIGNAL 131 --> SPARE
   // SIGNAL 132 --> SPARE
   // SIGNAL 133 --> SPARE
   // SIGNAL 134 --> SPARE
   // SIGNAL 135 --> SPARE
   // SIGNAL 136 --> SPARE
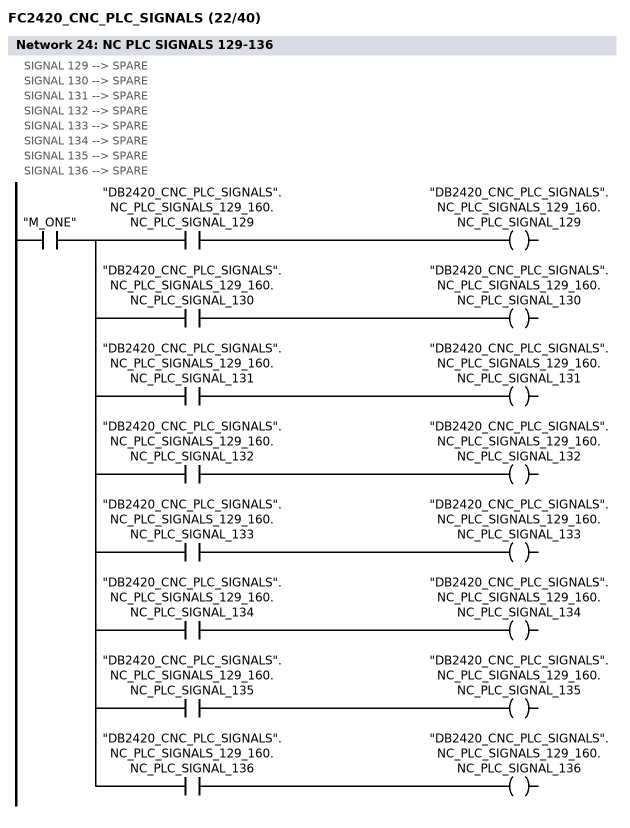
   RUNG wire#powerrail
      Contact( "M_ONE" )
      wire#w1
      Contact( "DB2420_CNC_PLC_SIGNALS".NC_PLC_SIGNALS_129_160.NC_PLC_SIGNAL_129 )
      Coil( "DB2420_CNC_PLC_SIGNALS".NC_PLC_SIGNALS_129_160.NC_PLC_SIGNAL_129 )
   END_RUNG
   RUNG wire#w1
      Contact( "DB2420_CNC_PLC_SIGNALS".NC_PLC_SIGNALS_129_160.NC_PLC_SIGNAL_130 )
      Coil( "DB2420_CNC_PLC_SIGNALS".NC_PLC_SIGNALS_129_160.NC_PLC_SIGNAL_130 )
   END_RUNG
   RUNG wire#w1
      Contact( "DB2420_CNC_PLC_SIGNALS".NC_PLC_SIGNALS_129_160.NC_PLC_SIGNAL_131 )
      Coil( "DB2420_CNC_PLC_SIGNALS".NC_PLC_SIGNALS_129_160.NC_PLC_SIGNAL_131 )
   END_RUNG
   RUNG wire#w1
      Contact( "DB2420_CNC_PLC_SIGNALS".NC_PLC_SIGNALS_129_160.NC_PLC_SIGNAL_132 )
      Coil( "DB2420_CNC_PLC_SIGNALS".NC_PLC_SIGNALS_129_160.NC_PLC_SIGNAL_132 )
   END_RUNG
   RUNG wire#w1
      Contact( "DB2420_CNC_PLC_SIGNALS".NC_PLC_SIGNALS_129_160.NC_PLC_SIGNAL_133 )
      Coil( "DB2420_CNC_PLC_SIGNALS".NC_PLC_SIGNALS_129_160.NC_PLC_SIGNAL_133 )
   END_RUNG
   RUNG wire#w1
      Contact( "DB2420_CNC_PLC_SIGNALS".NC_PLC_SIGNALS_129_160.NC_PLC_SIGNAL_134 )
      Coil( "DB2420_CNC_PLC_SIGNALS".NC_PLC_SIGNALS_129_160.NC_PLC_SIGNAL_134 )
   END_RUNG
   RUNG wire#w1
      Contact( "DB2420_CNC_PLC_SIGNALS".NC_PLC_SIGNALS_129_160.NC_PLC_SIGNAL_135 )
      Coil( "DB2420_CNC_PLC_SIGNALS".NC_PLC_SIGNALS_129_160.NC_PLC_SIGNAL_135 )
   END_RUNG
   RUNG wire#w1
      Contact( "DB2420_CNC_PLC_SIGNALS".NC_PLC_SIGNALS_129_160.NC_PLC_SIGNAL_136 )
      Coil( "DB2420_CNC_PLC_SIGNALS".NC_PLC_SIGNALS_129_160.NC_PLC_SIGNAL_136 )
   END_RUNG
   // the same network as SCL:
   "DB2420_CNC_PLC_SIGNALS".NC_PLC_SIGNALS_129_160.NC_PLC_SIGNAL_129 := "M_ONE" AND "DB2420_CNC_PLC_SIGNALS".NC_PLC_SIGNALS_129_160.NC_PLC_SIGNAL_129;
   "DB2420_CNC_PLC_SIGNALS".NC_PLC_SIGNALS_129_160.NC_PLC_SIGNAL_130 := "M_ONE" AND "DB2420_CNC_PLC_SIGNALS".NC_PLC_SIGNALS_129_160.NC_PLC_SIGNAL_130;
   "DB2420_CNC_PLC_SIGNALS".NC_PLC_SIGNALS_129_160.NC_PLC_SIGNAL_131 := "M_ONE" AND "DB2420_CNC_PLC_SIGNALS".NC_PLC_SIGNALS_129_160.NC_PLC_SIGNAL_131;
   "DB2420_CNC_PLC_SIGNALS".NC_PLC_SIGNALS_129_160.NC_PLC_SIGNAL_132 := "M_ONE" AND "DB2420_CNC_PLC_SIGNALS".NC_PLC_SIGNALS_129_160.NC_PLC_SIGNAL_132;
   "DB2420_CNC_PLC_SIGNALS".NC_PLC_SIGNALS_129_160.NC_PLC_SIGNAL_133 := "M_ONE" AND "DB2420_CNC_PLC_SIGNALS".NC_PLC_SIGNALS_129_160.NC_PLC_SIGNAL_133;
   "DB2420_CNC_PLC_SIGNALS".NC_PLC_SIGNALS_129_160.NC_PLC_SIGNAL_134 := "M_ONE" AND "DB2420_CNC_PLC_SIGNALS".NC_PLC_SIGNALS_129_160.NC_PLC_SIGNAL_134;
   "DB2420_CNC_PLC_SIGNALS".NC_PLC_SIGNALS_129_160.NC_PLC_SIGNAL_135 := "M_ONE" AND "DB2420_CNC_PLC_SIGNALS".NC_PLC_SIGNALS_129_160.NC_PLC_SIGNAL_135;
   "DB2420_CNC_PLC_SIGNALS".NC_PLC_SIGNALS_129_160.NC_PLC_SIGNAL_136 := "M_ONE" AND "DB2420_CNC_PLC_SIGNALS".NC_PLC_SIGNALS_129_160.NC_PLC_SIGNAL_136;
END_REGION

REGION Network 25: NC PLC SIGNALS 137-144
   // SIGNAL 137 --> SPARE
   // SIGNAL 138 --> SPARE
   // SIGNAL 139 --> SPARE
   // SIGNAL 140 --> SPARE
   // SIGNAL 141 --> SPARE
   // SIGNAL 142 --> SPARE
   // SIGNAL 143 --> SPARE
   // SIGNAL 144 --> SPARE
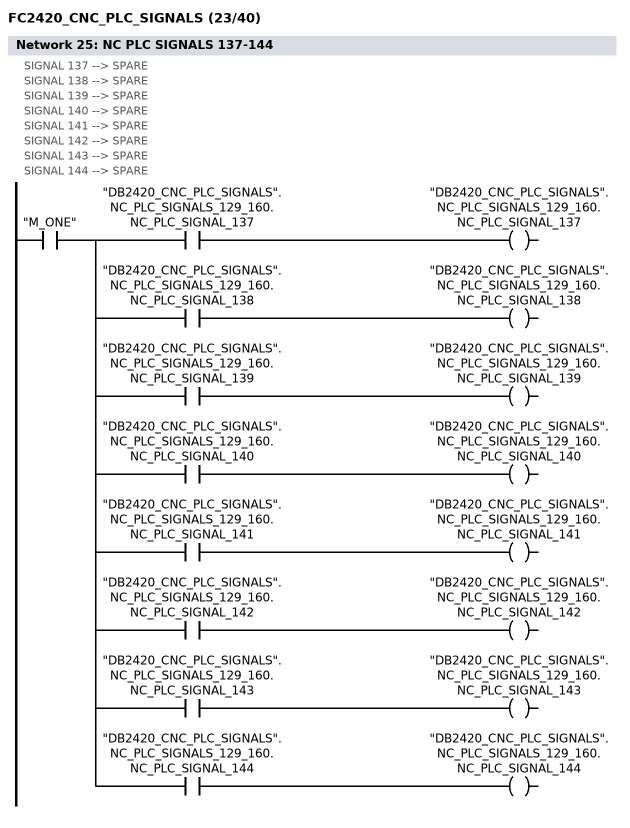
   RUNG wire#powerrail
      Contact( "M_ONE" )
      wire#w1
      Contact( "DB2420_CNC_PLC_SIGNALS".NC_PLC_SIGNALS_129_160.NC_PLC_SIGNAL_137 )
      Coil( "DB2420_CNC_PLC_SIGNALS".NC_PLC_SIGNALS_129_160.NC_PLC_SIGNAL_137 )
   END_RUNG
   RUNG wire#w1
      Contact( "DB2420_CNC_PLC_SIGNALS".NC_PLC_SIGNALS_129_160.NC_PLC_SIGNAL_138 )
      Coil( "DB2420_CNC_PLC_SIGNALS".NC_PLC_SIGNALS_129_160.NC_PLC_SIGNAL_138 )
   END_RUNG
   RUNG wire#w1
      Contact( "DB2420_CNC_PLC_SIGNALS".NC_PLC_SIGNALS_129_160.NC_PLC_SIGNAL_139 )
      Coil( "DB2420_CNC_PLC_SIGNALS".NC_PLC_SIGNALS_129_160.NC_PLC_SIGNAL_139 )
   END_RUNG
   RUNG wire#w1
      Contact( "DB2420_CNC_PLC_SIGNALS".NC_PLC_SIGNALS_129_160.NC_PLC_SIGNAL_140 )
      Coil( "DB2420_CNC_PLC_SIGNALS".NC_PLC_SIGNALS_129_160.NC_PLC_SIGNAL_140 )
   END_RUNG
   RUNG wire#w1
      Contact( "DB2420_CNC_PLC_SIGNALS".NC_PLC_SIGNALS_129_160.NC_PLC_SIGNAL_141 )
      Coil( "DB2420_CNC_PLC_SIGNALS".NC_PLC_SIGNALS_129_160.NC_PLC_SIGNAL_141 )
   END_RUNG
   RUNG wire#w1
      Contact( "DB2420_CNC_PLC_SIGNALS".NC_PLC_SIGNALS_129_160.NC_PLC_SIGNAL_142 )
      Coil( "DB2420_CNC_PLC_SIGNALS".NC_PLC_SIGNALS_129_160.NC_PLC_SIGNAL_142 )
   END_RUNG
   RUNG wire#w1
      Contact( "DB2420_CNC_PLC_SIGNALS".NC_PLC_SIGNALS_129_160.NC_PLC_SIGNAL_143 )
      Coil( "DB2420_CNC_PLC_SIGNALS".NC_PLC_SIGNALS_129_160.NC_PLC_SIGNAL_143 )
   END_RUNG
   RUNG wire#w1
      Contact( "DB2420_CNC_PLC_SIGNALS".NC_PLC_SIGNALS_129_160.NC_PLC_SIGNAL_144 )
      Coil( "DB2420_CNC_PLC_SIGNALS".NC_PLC_SIGNALS_129_160.NC_PLC_SIGNAL_144 )
   END_RUNG
   // the same network as SCL:
   "DB2420_CNC_PLC_SIGNALS".NC_PLC_SIGNALS_129_160.NC_PLC_SIGNAL_137 := "M_ONE" AND "DB2420_CNC_PLC_SIGNALS".NC_PLC_SIGNALS_129_160.NC_PLC_SIGNAL_137;
   "DB2420_CNC_PLC_SIGNALS".NC_PLC_SIGNALS_129_160.NC_PLC_SIGNAL_138 := "M_ONE" AND "DB2420_CNC_PLC_SIGNALS".NC_PLC_SIGNALS_129_160.NC_PLC_SIGNAL_138;
   "DB2420_CNC_PLC_SIGNALS".NC_PLC_SIGNALS_129_160.NC_PLC_SIGNAL_139 := "M_ONE" AND "DB2420_CNC_PLC_SIGNALS".NC_PLC_SIGNALS_129_160.NC_PLC_SIGNAL_139;
   "DB2420_CNC_PLC_SIGNALS".NC_PLC_SIGNALS_129_160.NC_PLC_SIGNAL_140 := "M_ONE" AND "DB2420_CNC_PLC_SIGNALS".NC_PLC_SIGNALS_129_160.NC_PLC_SIGNAL_140;
   "DB2420_CNC_PLC_SIGNALS".NC_PLC_SIGNALS_129_160.NC_PLC_SIGNAL_141 := "M_ONE" AND "DB2420_CNC_PLC_SIGNALS".NC_PLC_SIGNALS_129_160.NC_PLC_SIGNAL_141;
   "DB2420_CNC_PLC_SIGNALS".NC_PLC_SIGNALS_129_160.NC_PLC_SIGNAL_142 := "M_ONE" AND "DB2420_CNC_PLC_SIGNALS".NC_PLC_SIGNALS_129_160.NC_PLC_SIGNAL_142;
   "DB2420_CNC_PLC_SIGNALS".NC_PLC_SIGNALS_129_160.NC_PLC_SIGNAL_143 := "M_ONE" AND "DB2420_CNC_PLC_SIGNALS".NC_PLC_SIGNALS_129_160.NC_PLC_SIGNAL_143;
   "DB2420_CNC_PLC_SIGNALS".NC_PLC_SIGNALS_129_160.NC_PLC_SIGNAL_144 := "M_ONE" AND "DB2420_CNC_PLC_SIGNALS".NC_PLC_SIGNALS_129_160.NC_PLC_SIGNAL_144;
END_REGION

REGION Network 26: NC PLC SIGNALS 145-152
   // SIGNAL 145 --> SPARE
   // SIGNAL 146 --> SPARE
   // SIGNAL 147 --> SPARE
   // SIGNAL 148 --> SPARE
   // SIGNAL 149 --> SPARE
   // SIGNAL 150 --> SPARE
   // SIGNAL 151 --> SPARE
   // SIGNAL 152 --> SPARE
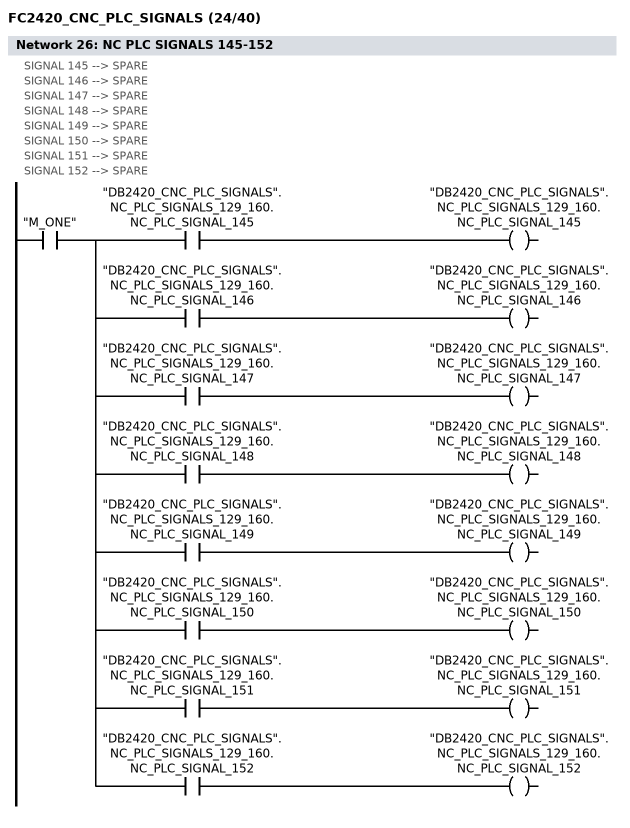
   RUNG wire#powerrail
      Contact( "M_ONE" )
      wire#w1
      Contact( "DB2420_CNC_PLC_SIGNALS".NC_PLC_SIGNALS_129_160.NC_PLC_SIGNAL_145 )
      Coil( "DB2420_CNC_PLC_SIGNALS".NC_PLC_SIGNALS_129_160.NC_PLC_SIGNAL_145 )
   END_RUNG
   RUNG wire#w1
      Contact( "DB2420_CNC_PLC_SIGNALS".NC_PLC_SIGNALS_129_160.NC_PLC_SIGNAL_146 )
      Coil( "DB2420_CNC_PLC_SIGNALS".NC_PLC_SIGNALS_129_160.NC_PLC_SIGNAL_146 )
   END_RUNG
   RUNG wire#w1
      Contact( "DB2420_CNC_PLC_SIGNALS".NC_PLC_SIGNALS_129_160.NC_PLC_SIGNAL_147 )
      Coil( "DB2420_CNC_PLC_SIGNALS".NC_PLC_SIGNALS_129_160.NC_PLC_SIGNAL_147 )
   END_RUNG
   RUNG wire#w1
      Contact( "DB2420_CNC_PLC_SIGNALS".NC_PLC_SIGNALS_129_160.NC_PLC_SIGNAL_148 )
      Coil( "DB2420_CNC_PLC_SIGNALS".NC_PLC_SIGNALS_129_160.NC_PLC_SIGNAL_148 )
   END_RUNG
   RUNG wire#w1
      Contact( "DB2420_CNC_PLC_SIGNALS".NC_PLC_SIGNALS_129_160.NC_PLC_SIGNAL_149 )
      Coil( "DB2420_CNC_PLC_SIGNALS".NC_PLC_SIGNALS_129_160.NC_PLC_SIGNAL_149 )
   END_RUNG
   RUNG wire#w1
      Contact( "DB2420_CNC_PLC_SIGNALS".NC_PLC_SIGNALS_129_160.NC_PLC_SIGNAL_150 )
      Coil( "DB2420_CNC_PLC_SIGNALS".NC_PLC_SIGNALS_129_160.NC_PLC_SIGNAL_150 )
   END_RUNG
   RUNG wire#w1
      Contact( "DB2420_CNC_PLC_SIGNALS".NC_PLC_SIGNALS_129_160.NC_PLC_SIGNAL_151 )
      Coil( "DB2420_CNC_PLC_SIGNALS".NC_PLC_SIGNALS_129_160.NC_PLC_SIGNAL_151 )
   END_RUNG
   RUNG wire#w1
      Contact( "DB2420_CNC_PLC_SIGNALS".NC_PLC_SIGNALS_129_160.NC_PLC_SIGNAL_152 )
      Coil( "DB2420_CNC_PLC_SIGNALS".NC_PLC_SIGNALS_129_160.NC_PLC_SIGNAL_152 )
   END_RUNG
   // the same network as SCL:
   "DB2420_CNC_PLC_SIGNALS".NC_PLC_SIGNALS_129_160.NC_PLC_SIGNAL_145 := "M_ONE" AND "DB2420_CNC_PLC_SIGNALS".NC_PLC_SIGNALS_129_160.NC_PLC_SIGNAL_145;
   "DB2420_CNC_PLC_SIGNALS".NC_PLC_SIGNALS_129_160.NC_PLC_SIGNAL_146 := "M_ONE" AND "DB2420_CNC_PLC_SIGNALS".NC_PLC_SIGNALS_129_160.NC_PLC_SIGNAL_146;
   "DB2420_CNC_PLC_SIGNALS".NC_PLC_SIGNALS_129_160.NC_PLC_SIGNAL_147 := "M_ONE" AND "DB2420_CNC_PLC_SIGNALS".NC_PLC_SIGNALS_129_160.NC_PLC_SIGNAL_147;
   "DB2420_CNC_PLC_SIGNALS".NC_PLC_SIGNALS_129_160.NC_PLC_SIGNAL_148 := "M_ONE" AND "DB2420_CNC_PLC_SIGNALS".NC_PLC_SIGNALS_129_160.NC_PLC_SIGNAL_148;
   "DB2420_CNC_PLC_SIGNALS".NC_PLC_SIGNALS_129_160.NC_PLC_SIGNAL_149 := "M_ONE" AND "DB2420_CNC_PLC_SIGNALS".NC_PLC_SIGNALS_129_160.NC_PLC_SIGNAL_149;
   "DB2420_CNC_PLC_SIGNALS".NC_PLC_SIGNALS_129_160.NC_PLC_SIGNAL_150 := "M_ONE" AND "DB2420_CNC_PLC_SIGNALS".NC_PLC_SIGNALS_129_160.NC_PLC_SIGNAL_150;
   "DB2420_CNC_PLC_SIGNALS".NC_PLC_SIGNALS_129_160.NC_PLC_SIGNAL_151 := "M_ONE" AND "DB2420_CNC_PLC_SIGNALS".NC_PLC_SIGNALS_129_160.NC_PLC_SIGNAL_151;
   "DB2420_CNC_PLC_SIGNALS".NC_PLC_SIGNALS_129_160.NC_PLC_SIGNAL_152 := "M_ONE" AND "DB2420_CNC_PLC_SIGNALS".NC_PLC_SIGNALS_129_160.NC_PLC_SIGNAL_152;
END_REGION

REGION Network 27: NC PLC SIGNALS 153-160
   // SIGNAL 153 --> SPARE
   // SIGNAL 154 --> SPARE
   // SIGNAL 155 --> SPARE
   // SIGNAL 156 --> SPARE
   // SIGNAL 157 --> SPARE
   // SIGNAL 158 --> SPARE
   // SIGNAL 159 --> SPARE
   // SIGNAL 160 --> SPARE
